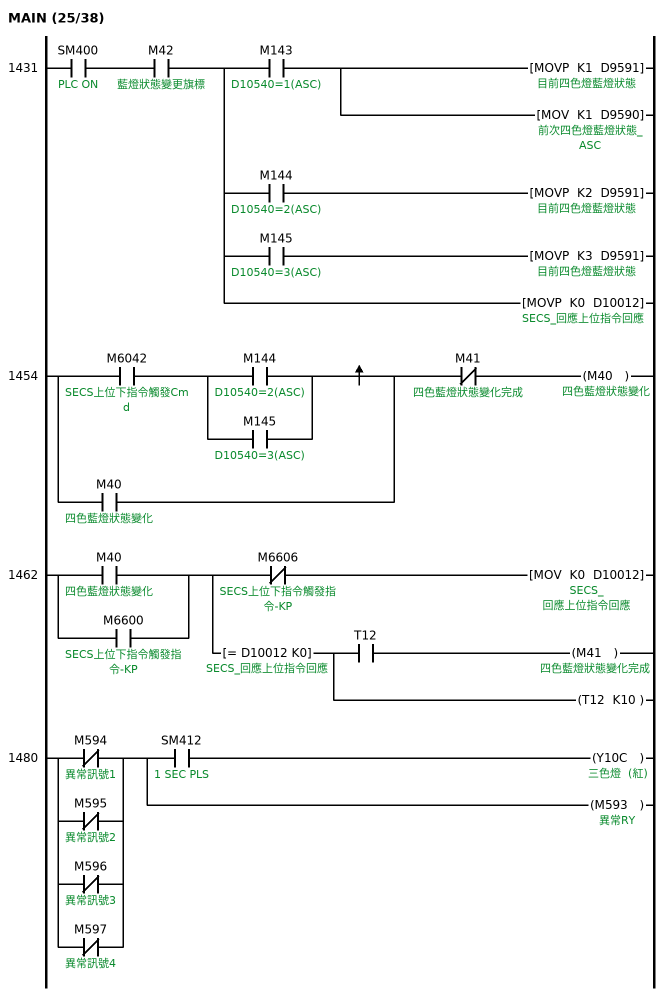
[picture p24: ladder of MAIN, rungs at steps 1431 to 1480]
1431  LD      SM400  ; PLC ON
      AND     M42  ; 藍燈狀態變更旗標
      MPS
      AND     M143  ; D10540=1(ASC)
      MOVP    K1 D9591
      MOV     K1 D9590
      MRD
      AND     M144  ; D10540=2(ASC)
      MOVP    K2 D9591
      MRD
      AND     M145  ; D10540=3(ASC)
      MOVP    K3 D9591
      MPP
      MOVP    K0 D10012  ; SECS_回應上位指令回應
1454  LD      M6042  ; SECS上位下指令觸發Cmd
      LD      M144  ; D10540=2(ASC)
      OR      M145  ; D10540=3(ASC)
      ANB
      MEP
      OR      M40  ; 四色藍燈狀態變化
      ANI     M41  ; 四色藍燈狀態變化完成
      OUT     M40  ; 四色藍燈狀態變化
1462  LD      M40  ; 四色藍燈狀態變化
      OR      M6600  ; SECS上位下指令觸發指令-KP
      MPS
      ANI     M6606  ; SECS上位下指令觸發指令-KP
      MOV     K0 D10012
      MPP
      AND=    D10012 K0  ; SECS_回應上位指令回應
      MPS
      AND     T12
      OUT     M41  ; 四色藍燈狀態變化完成
      MPP
      OUT     T12 K10
1480  LDI     M594  ; 異常訊號1
      ORI     M595  ; 異常訊號2
      ORI     M596  ; 異常訊號3
      ORI     M597  ; 異常訊號4
      MPS
      AND     SM412  ; 1 SEC PLS
      OUT     Y10C  ; 三色燈  (紅)
      MPP
      OUT     M593  ; 異常RY
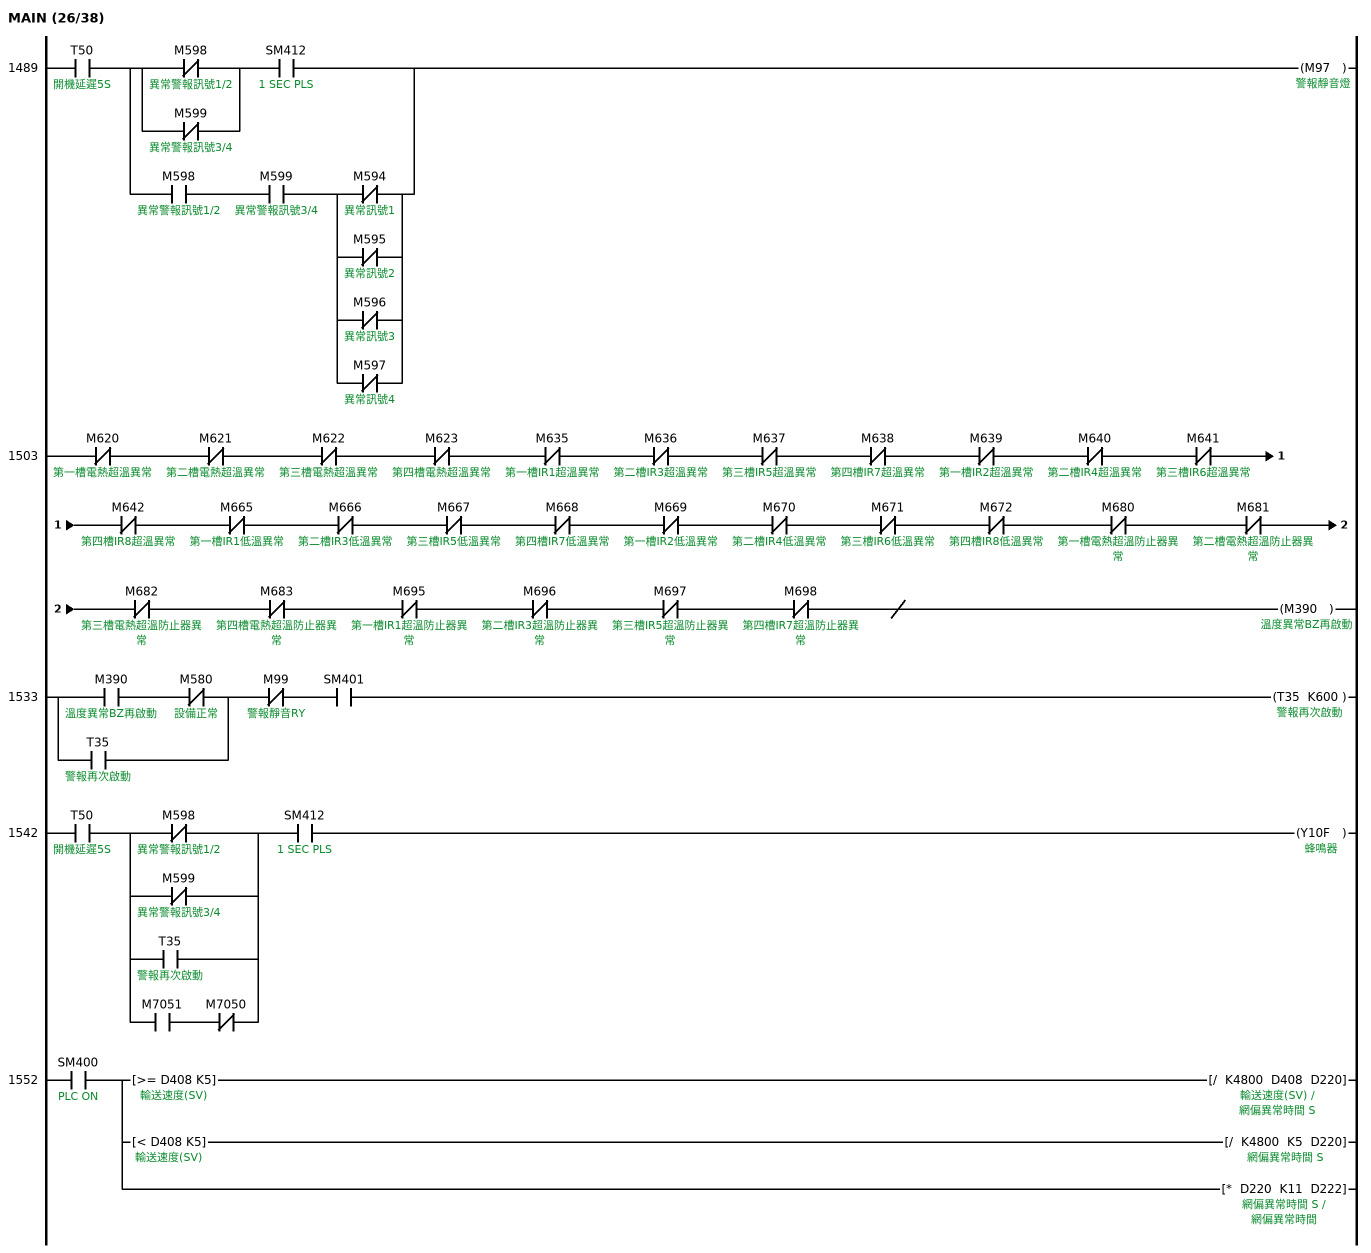
1489  LD      T50  ; 開機延遲5S
      LDI     M598  ; 異常警報訊號1/2
      ORI     M599  ; 異常警報訊號3/4
      AND     SM412  ; 1 SEC PLS
      LD      M598  ; 異常警報訊號1/2
      AND     M599  ; 異常警報訊號3/4
      LDI     M594  ; 異常訊號1
      ORI     M595  ; 異常訊號2
      ORI     M596  ; 異常訊號3
      ORI     M597  ; 異常訊號4
      ANB
      ORB
      ANB
      OUT     M97  ; 警報靜音燈
1503  LDI     M620  ; 第一槽電熱超溫異常
      ANI     M621  ; 第二槽電熱超溫異常
      ANI     M622  ; 第三槽電熱超溫異常
      ANI     M623  ; 第四槽電熱超溫異常
      ANI     M635  ; 第一槽IR1超溫異常
      ANI     M636  ; 第二槽IR3超溫異常
      ANI     M637  ; 第三槽IR5超溫異常
      ANI     M638  ; 第四槽IR7超溫異常
      ANI     M639  ; 第一槽IR2超溫異常
      ANI     M640  ; 第二槽IR4超溫異常
      ANI     M641  ; 第三槽IR6超溫異常
      ANI     M642  ; 第四槽IR8超溫異常
      ANI     M665  ; 第一槽IR1低溫異常
      ANI     M666  ; 第二槽IR3低溫異常
      ANI     M667  ; 第三槽IR5低溫異常
      ANI     M668  ; 第四槽IR7低溫異常
      ANI     M669  ; 第一槽IR2低溫異常
      ANI     M670  ; 第二槽IR4低溫異常
      ANI     M671  ; 第三槽IR6低溫異常
      ANI     M672  ; 第四槽IR8低溫異常
      ANI     M680  ; 第一槽電熱超溫防止器異常
      ANI     M681  ; 第二槽電熱超溫防止器異常
      ANI     M682  ; 第三槽電熱超溫防止器異常
      ANI     M683  ; 第四槽電熱超溫防止器異常
      ANI     M695  ; 第一槽IR1超溫防止器異常
      ANI     M696  ; 第二槽IR3超溫防止器異常
      ANI     M697  ; 第三槽IR5超溫防止器異常
      ANI     M698  ; 第四槽IR7超溫防止器異常
      INV
      OUT     M390  ; 溫度異常BZ再啟動
1533  LD      M390  ; 溫度異常BZ再啟動
      ANI     M580  ; 設備正常
      OR      T35  ; 警報再次啟動
      ANI     M99  ; 警報靜音RY
      AND     SM401
      OUT     T35 K600  ; 警報再次啟動
1542  LD      T50  ; 開機延遲5S
      LDI     M598  ; 異常警報訊號1/2
      ORI     M599  ; 異常警報訊號3/4
      OR      T35  ; 警報再次啟動
      LD      M7051
      ANI     M7050
      ORB
      ANB
      AND     SM412  ; 1 SEC PLS
      OUT     Y10F  ; 蜂鳴器
1552  LD      SM400  ; PLC ON
      MPS
      AND>=   D408 K5  ; 輸送速度(SV)
      /       K4800 D408 D220  ; 網偏異常時間 S
      MRD
      AND<    D408 K5  ; 輸送速度(SV)
      /       K4800 K5 D220
      MPP
      *       D220 K11 D222  ; 網偏異常時間
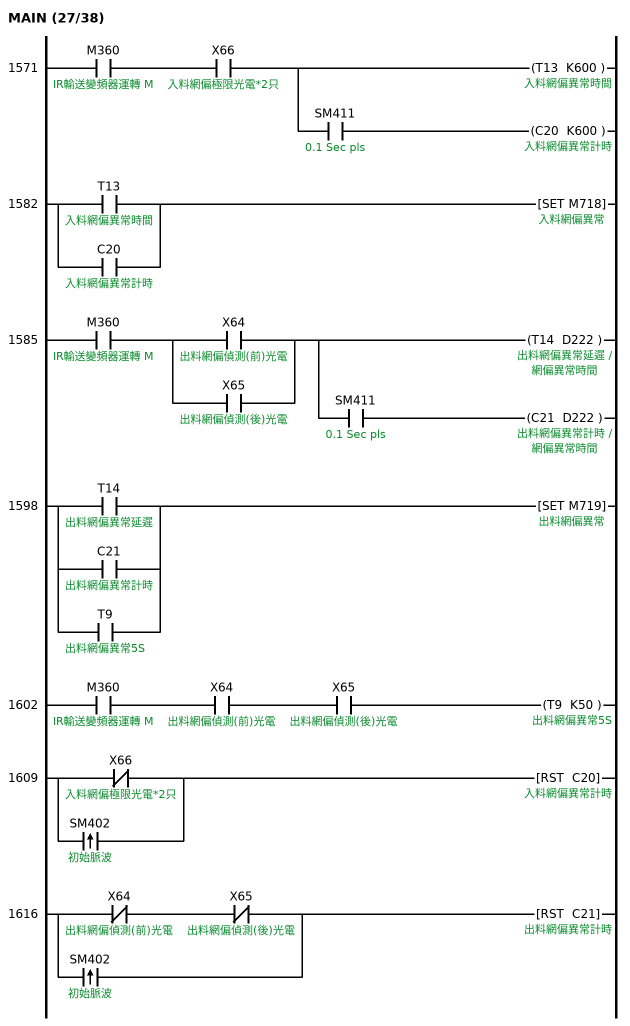
1571  LD      M360  ; IR輸送變頻器運轉 M
      AND     X66  ; 入料網偏極限光電*2只
      OUT     T13 K600  ; 入料網偏異常時間
      AND     SM411  ; 0.1 Sec pls
      OUT     C20 K600  ; 入料網偏異常計時
1582  LD      T13  ; 入料網偏異常時間
      OR      C20  ; 入料網偏異常計時
      SET     M718  ; 入料網偏異常
1585  LD      M360  ; IR輸送變頻器運轉 M
      LD      X64  ; 出料網偏偵測(前)光電
      OR      X65  ; 出料網偏偵測(後)光電
      ANB
      OUT     T14 D222  ; 出料網偏異常延遲 / 網偏異常時間
      AND     SM411  ; 0.1 Sec pls
      OUT     C21 D222  ; 出料網偏異常計時 / 網偏異常時間
1598  LD      T14  ; 出料網偏異常延遲
      OR      C21  ; 出料網偏異常計時
      OR      T9  ; 出料網偏異常5S
      SET     M719  ; 出料網偏異常
1602  LD      M360  ; IR輸送變頻器運轉 M
      AND     X64  ; 出料網偏偵測(前)光電
      AND     X65  ; 出料網偏偵測(後)光電
      OUT     T9 K50  ; 出料網偏異常5S
1609  LDI     X66  ; 入料網偏極限光電*2只
      ORP     SM402  ; 初始脈波
      RST     C20  ; 入料網偏異常計時
1616  LDI     X64  ; 出料網偏偵測(前)光電
      ANI     X65  ; 出料網偏偵測(後)光電
      ORP     SM402  ; 初始脈波
      RST     C21  ; 出料網偏異常計時
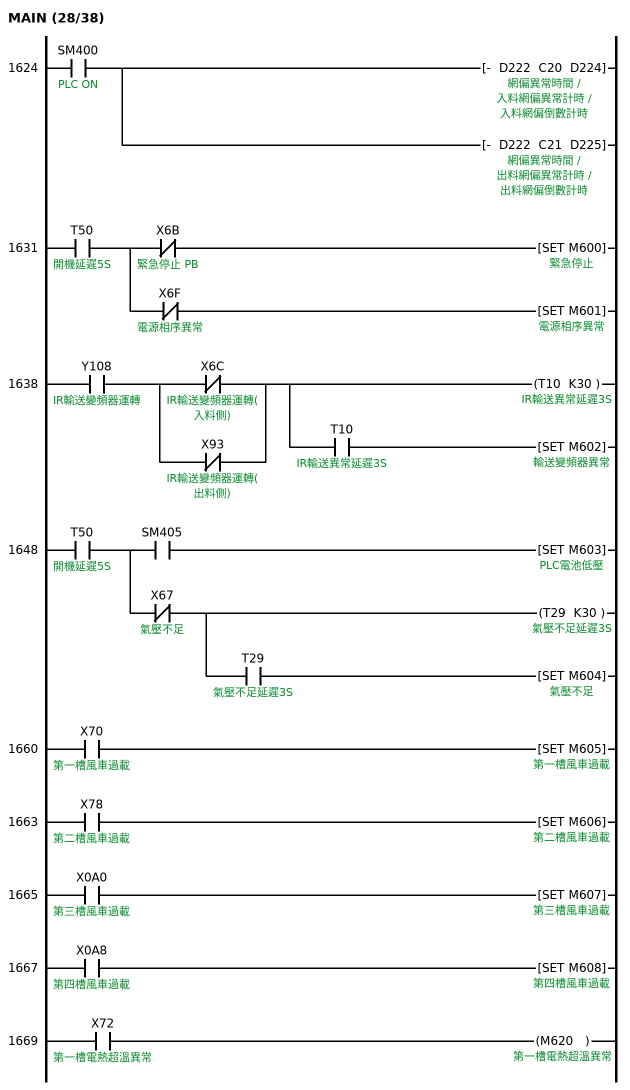
1624  LD      SM400  ; PLC ON
      -       D222 C20 D224  ; 入料網偏倒數計時
      -       D222 C21 D225  ; 出料網偏倒數計時
1631  LD      T50  ; 開機延遲5S
      MPS
      ANI     X6B  ; 緊急停止 PB
      SET     M600  ; 緊急停止
      MPP
      ANI     X6F  ; 電源相序異常
      SET     M601  ; 電源相序異常
1638  LD      Y108  ; IR輸送變頻器運轉
      LDI     X6C  ; IR輸送變頻器運轉(入料側)
      ORI     X93  ; IR輸送變頻器運轉(出料側)
      ANB
      OUT     T10 K30  ; IR輸送異常延遲3S
      AND     T10  ; IR輸送異常延遲3S
      SET     M602  ; 輸送變頻器異常
1648  LD      T50  ; 開機延遲5S
      MPS
      AND     SM405
      SET     M603  ; PLC電池低壓
      MPP
      ANI     X67  ; 氣壓不足
      OUT     T29 K30  ; 氣壓不足延遲3S
      AND     T29  ; 氣壓不足延遲3S
      SET     M604  ; 氣壓不足
1660  LD      X70  ; 第一槽風車過載
      SET     M605  ; 第一槽風車過載
        [note] 
1663  LD      X78  ; 第二槽風車過載
      SET     M606  ; 第二槽風車過載
1665  LD      X0A0  ; 第三槽風車過載
      SET     M607  ; 第三槽風車過載
1667  LD      X0A8  ; 第四槽風車過載
      SET     M608  ; 第四槽風車過載
1669  LD      X72  ; 第一槽電熱超溫異常
      OUT     M620  ; 第一槽電熱超溫異常
        [note] 
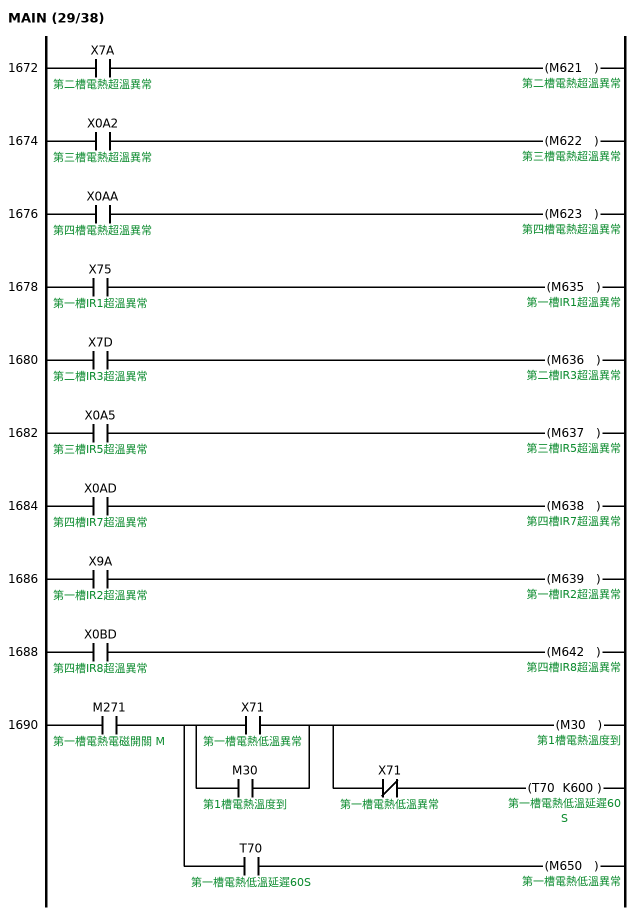
1672  LD      X7A  ; 第二槽電熱超溫異常
      OUT     M621  ; 第二槽電熱超溫異常
1674  LD      X0A2  ; 第三槽電熱超溫異常
      OUT     M622  ; 第三槽電熱超溫異常
1676  LD      X0AA  ; 第四槽電熱超溫異常
      OUT     M623  ; 第四槽電熱超溫異常
1678  LD      X75  ; 第一槽IR1超溫異常
      OUT     M635  ; 第一槽IR1超溫異常
1680  LD      X7D  ; 第二槽IR3超溫異常
      OUT     M636  ; 第二槽IR3超溫異常
1682  LD      X0A5  ; 第三槽IR5超溫異常
      OUT     M637  ; 第三槽IR5超溫異常
1684  LD      X0AD  ; 第四槽IR7超溫異常
      OUT     M638  ; 第四槽IR7超溫異常
1686  LD      X9A  ; 第一槽IR2超溫異常
      OUT     M639  ; 第一槽IR2超溫異常
1688  LD      X0BD  ; 第四槽IR8超溫異常
      OUT     M642  ; 第四槽IR8超溫異常
1690  LD      M271  ; 第一槽電熱電磁開關 M
      MPS
      LD      X71  ; 第一槽電熱低溫異常
      OR      M30  ; 第1槽電熱溫度到
      ANB
      OUT     M30  ; 第1槽電熱溫度到
        [note] 
      ANI     X71  ; 第一槽電熱低溫異常
      OUT     T70 K600  ; 第一槽電熱低溫延遲60S
      MPP
      AND     T70  ; 第一槽電熱低溫延遲60S
      OUT     M650  ; 第一槽電熱低溫異常
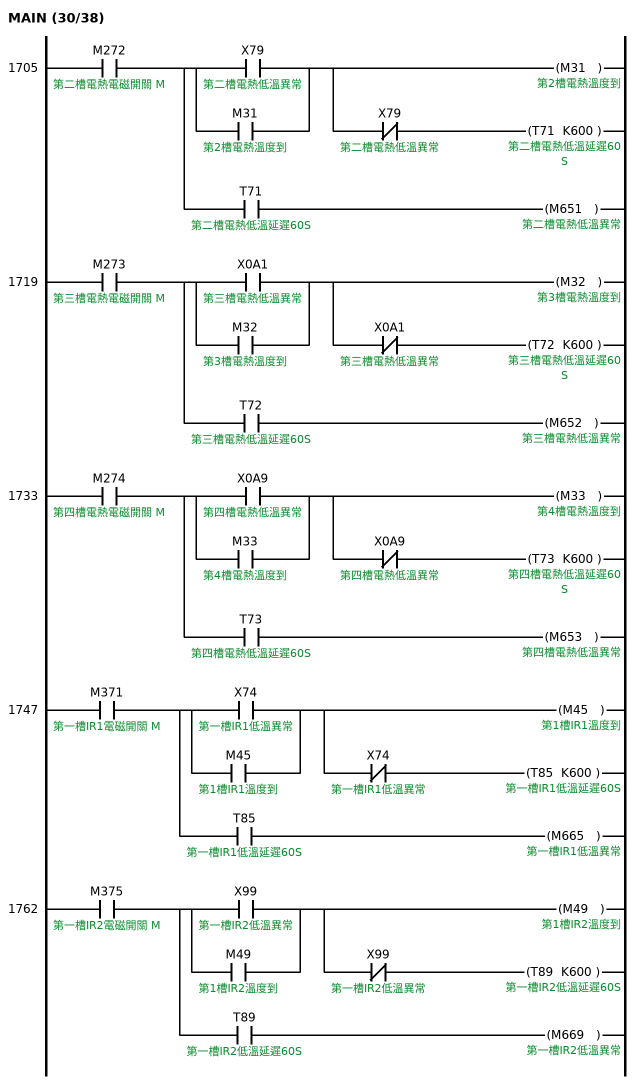
1705  LD      M272  ; 第二槽電熱電磁開關 M
      MPS
      LD      X79  ; 第二槽電熱低溫異常
      OR      M31  ; 第2槽電熱溫度到
      ANB
      OUT     M31  ; 第2槽電熱溫度到
      ANI     X79  ; 第二槽電熱低溫異常
      OUT     T71 K600  ; 第二槽電熱低溫延遲60S
      MPP
      AND     T71  ; 第二槽電熱低溫延遲60S
      OUT     M651  ; 第二槽電熱低溫異常
1719  LD      M273  ; 第三槽電熱電磁開關 M
      MPS
      LD      X0A1  ; 第三槽電熱低溫異常
      OR      M32  ; 第3槽電熱溫度到
      ANB
      OUT     M32  ; 第3槽電熱溫度到
      ANI     X0A1  ; 第三槽電熱低溫異常
      OUT     T72 K600  ; 第三槽電熱低溫延遲60S
      MPP
      AND     T72  ; 第三槽電熱低溫延遲60S
      OUT     M652  ; 第三槽電熱低溫異常
1733  LD      M274  ; 第四槽電熱電磁開關 M
      MPS
      LD      X0A9  ; 第四槽電熱低溫異常
      OR      M33  ; 第4槽電熱溫度到
      ANB
      OUT     M33  ; 第4槽電熱溫度到
      ANI     X0A9  ; 第四槽電熱低溫異常
      OUT     T73 K600  ; 第四槽電熱低溫延遲60S
      MPP
      AND     T73  ; 第四槽電熱低溫延遲60S
      OUT     M653  ; 第四槽電熱低溫異常
1747  LD      M371  ; 第一槽IR1電磁開關 M
      MPS
      LD      X74  ; 第一槽IR1低溫異常
      OR      M45  ; 第1槽IR1溫度到
      ANB
      OUT     M45  ; 第1槽IR1溫度到
        [note] 
      ANI     X74  ; 第一槽IR1低溫異常
      OUT     T85 K600  ; 第一槽IR1低溫延遲60S
      MPP
      AND     T85  ; 第一槽IR1低溫延遲60S
      OUT     M665  ; 第一槽IR1低溫異常
1762  LD      M375  ; 第一槽IR2電磁開關 M
      MPS
      LD      X99  ; 第一槽IR2低溫異常
      OR      M49  ; 第1槽IR2溫度到
      ANB
      OUT     M49  ; 第1槽IR2溫度到
      ANI     X99  ; 第一槽IR2低溫異常
      OUT     T89 K600  ; 第一槽IR2低溫延遲60S
      MPP
      AND     T89  ; 第一槽IR2低溫延遲60S
      OUT     M669  ; 第一槽IR2低溫異常
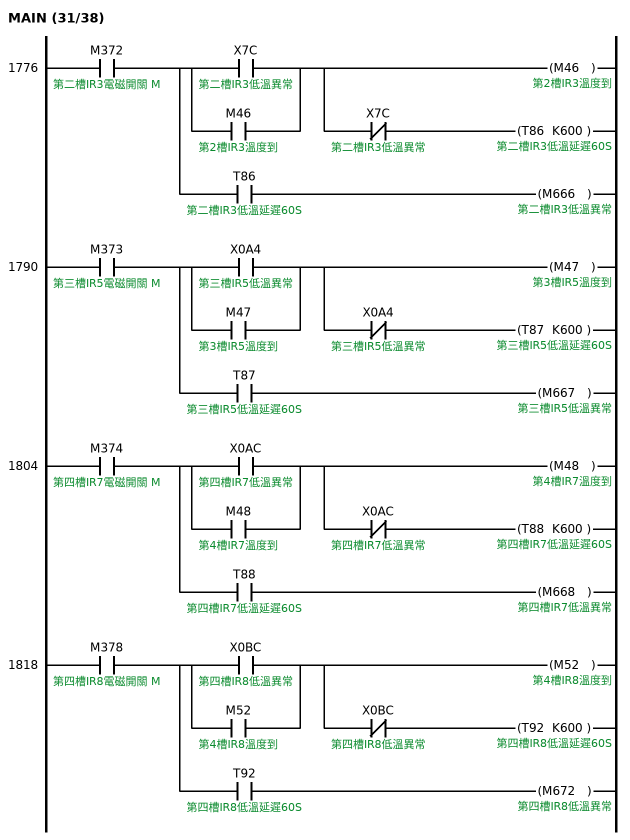
1776  LD      M372  ; 第二槽IR3電磁開關 M
      MPS
      LD      X7C  ; 第二槽IR3低溫異常
      OR      M46  ; 第2槽IR3溫度到
      ANB
      OUT     M46  ; 第2槽IR3溫度到
      ANI     X7C  ; 第二槽IR3低溫異常
      OUT     T86 K600  ; 第二槽IR3低溫延遲60S
      MPP
      AND     T86  ; 第二槽IR3低溫延遲60S
      OUT     M666  ; 第二槽IR3低溫異常
1790  LD      M373  ; 第三槽IR5電磁開關 M
      MPS
      LD      X0A4  ; 第三槽IR5低溫異常
      OR      M47  ; 第3槽IR5溫度到
      ANB
      OUT     M47  ; 第3槽IR5溫度到
      ANI     X0A4  ; 第三槽IR5低溫異常
      OUT     T87 K600  ; 第三槽IR5低溫延遲60S
      MPP
      AND     T87  ; 第三槽IR5低溫延遲60S
      OUT     M667  ; 第三槽IR5低溫異常
1804  LD      M374  ; 第四槽IR7電磁開關 M
      MPS
      LD      X0AC  ; 第四槽IR7低溫異常
      OR      M48  ; 第4槽IR7溫度到
      ANB
      OUT     M48  ; 第4槽IR7溫度到
      ANI     X0AC  ; 第四槽IR7低溫異常
      OUT     T88 K600  ; 第四槽IR7低溫延遲60S
      MPP
      AND     T88  ; 第四槽IR7低溫延遲60S
      OUT     M668  ; 第四槽IR7低溫異常
1818  LD      M378  ; 第四槽IR8電磁開關 M
      MPS
      LD      X0BC  ; 第四槽IR8低溫異常
      OR      M52  ; 第4槽IR8溫度到
      ANB
      OUT     M52  ; 第4槽IR8溫度到
      ANI     X0BC  ; 第四槽IR8低溫異常
      OUT     T92 K600  ; 第四槽IR8低溫延遲60S
      MPP
      AND     T92  ; 第四槽IR8低溫延遲60S
      OUT     M672  ; 第四槽IR8低溫異常
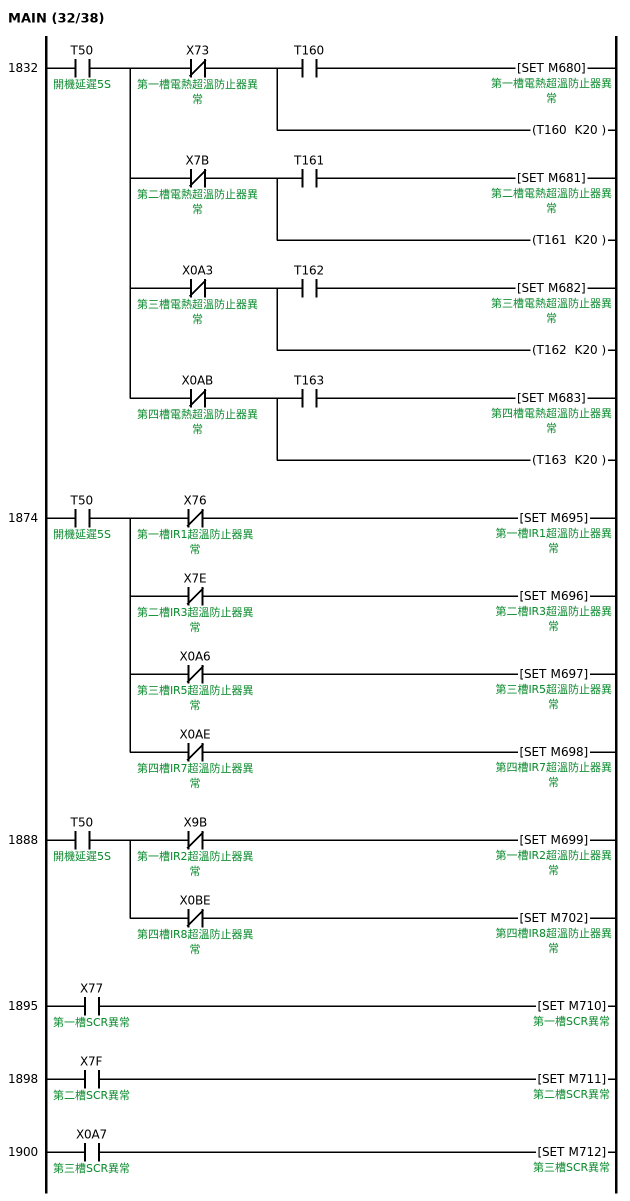
1832  LD      T50  ; 開機延遲5S
      MPS
      ANI     X73  ; 第一槽電熱超溫防止器異常
      MPS
      AND     T160
      SET     M680  ; 第一槽電熱超溫防止器異常
        [note] 
      MPP
      OUT     T160 K20
      MRD
      ANI     X7B  ; 第二槽電熱超溫防止器異常
      MPS
      AND     T161
      SET     M681  ; 第二槽電熱超溫防止器異常
      MPP
      OUT     T161 K20
      MRD
      ANI     X0A3  ; 第三槽電熱超溫防止器異常
      MPS
      AND     T162
      SET     M682  ; 第三槽電熱超溫防止器異常
      MPP
      OUT     T162 K20
      MPP
      ANI     X0AB  ; 第四槽電熱超溫防止器異常
      MPS
      AND     T163
      SET     M683  ; 第四槽電熱超溫防止器異常
      MPP
      OUT     T163 K20
1874  LD      T50  ; 開機延遲5S
      MPS
      ANI     X76  ; 第一槽IR1超溫防止器異常
      SET     M695  ; 第一槽IR1超溫防止器異常
        [note] 
      MRD
      ANI     X7E  ; 第二槽IR3超溫防止器異常
      SET     M696  ; 第二槽IR3超溫防止器異常
      MRD
      ANI     X0A6  ; 第三槽IR5超溫防止器異常
      SET     M697  ; 第三槽IR5超溫防止器異常
      MPP
      ANI     X0AE  ; 第四槽IR7超溫防止器異常
      SET     M698  ; 第四槽IR7超溫防止器異常
1888  LD      T50  ; 開機延遲5S
      MPS
      ANI     X9B  ; 第一槽IR2超溫防止器異常
      SET     M699  ; 第一槽IR2超溫防止器異常
      MPP
      ANI     X0BE  ; 第四槽IR8超溫防止器異常
      SET     M702  ; 第四槽IR8超溫防止器異常
1895  LD      X77  ; 第一槽SCR異常
      SET     M710  ; 第一槽SCR異常
        [note] 
1898  LD      X7F  ; 第二槽SCR異常
      SET     M711  ; 第二槽SCR異常
1900  LD      X0A7  ; 第三槽SCR異常
      SET     M712  ; 第三槽SCR異常
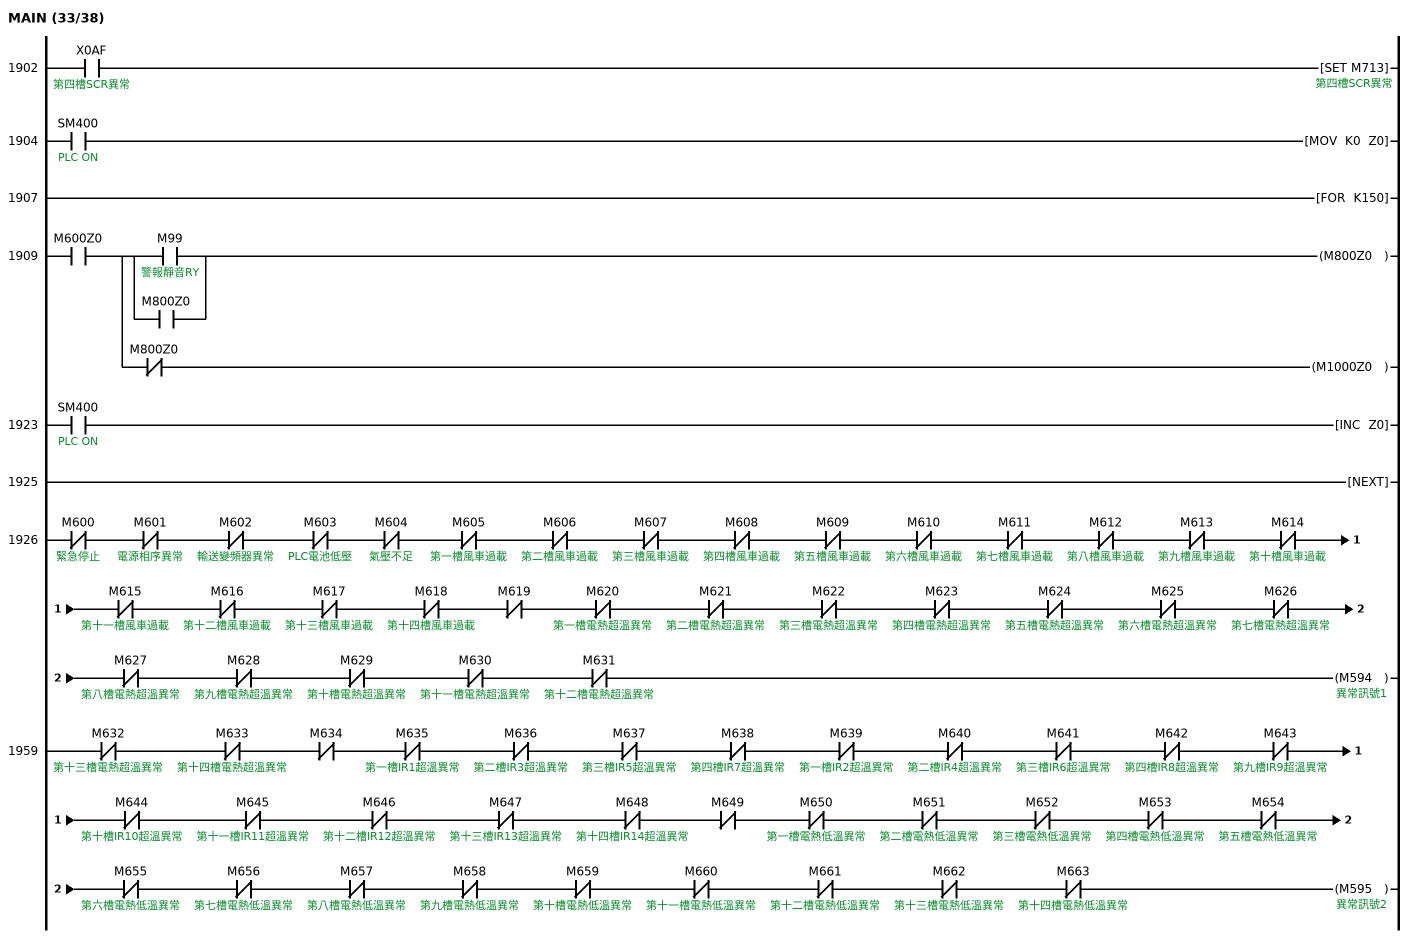
1902  LD      X0AF  ; 第四槽SCR異常
      SET     M713  ; 第四槽SCR異常
1904  LD      SM400  ; PLC ON
      MOV     K0 Z0
1907  FOR     K150
1909  LD      M600Z0
      MPS
      LD      M99  ; 警報靜音RY
      OR      M800Z0
      ANB
      OUT     M800Z0
      MPP
      ANI     M800Z0
      OUT     M1000Z0
1923  LD      SM400  ; PLC ON
      INC     Z0
1925  NEXT
1926  LDI     M600  ; 緊急停止
      ANI     M601  ; 電源相序異常
      ANI     M602  ; 輸送變頻器異常
      ANI     M603  ; PLC電池低壓
      ANI     M604  ; 氣壓不足
      ANI     M605  ; 第一槽風車過載
      ANI     M606  ; 第二槽風車過載
      ANI     M607  ; 第三槽風車過載
      ANI     M608  ; 第四槽風車過載
      ANI     M609  ; 第五槽風車過載
      ANI     M610  ; 第六槽風車過載
      ANI     M611  ; 第七槽風車過載
      ANI     M612  ; 第八槽風車過載
      ANI     M613  ; 第九槽風車過載
      ANI     M614  ; 第十槽風車過載
      ANI     M615  ; 第十一槽風車過載
      ANI     M616  ; 第十二槽風車過載
      ANI     M617  ; 第十三槽風車過載
      ANI     M618  ; 第十四槽風車過載
      ANI     M619
      ANI     M620  ; 第一槽電熱超溫異常
      ANI     M621  ; 第二槽電熱超溫異常
      ANI     M622  ; 第三槽電熱超溫異常
      ANI     M623  ; 第四槽電熱超溫異常
      ANI     M624  ; 第五槽電熱超溫異常
      ANI     M625  ; 第六槽電熱超溫異常
      ANI     M626  ; 第七槽電熱超溫異常
      ANI     M627  ; 第八槽電熱超溫異常
      ANI     M628  ; 第九槽電熱超溫異常
      ANI     M629  ; 第十槽電熱超溫異常
      ANI     M630  ; 第十一槽電熱超溫異常
      ANI     M631  ; 第十二槽電熱超溫異常
      OUT     M594  ; 異常訊號1
1959  LDI     M632  ; 第十三槽電熱超溫異常
      ANI     M633  ; 第十四槽電熱超溫異常
      ANI     M634
      ANI     M635  ; 第一槽IR1超溫異常
      ANI     M636  ; 第二槽IR3超溫異常
      ANI     M637  ; 第三槽IR5超溫異常
      ANI     M638  ; 第四槽IR7超溫異常
      ANI     M639  ; 第一槽IR2超溫異常
      ANI     M640  ; 第二槽IR4超溫異常
      ANI     M641  ; 第三槽IR6超溫異常
      ANI     M642  ; 第四槽IR8超溫異常
      ANI     M643  ; 第九槽IR9超溫異常
      ANI     M644  ; 第十槽IR10超溫異常
      ANI     M645  ; 第十一槽IR11超溫異常
      ANI     M646  ; 第十二槽IR12超溫異常
      ANI     M647  ; 第十三槽IR13超溫異常
      ANI     M648  ; 第十四槽IR14超溫異常
      ANI     M649
      ANI     M650  ; 第一槽電熱低溫異常
      ANI     M651  ; 第二槽電熱低溫異常
      ANI     M652  ; 第三槽電熱低溫異常
      ANI     M653  ; 第四槽電熱低溫異常
      ANI     M654  ; 第五槽電熱低溫異常
      ANI     M655  ; 第六槽電熱低溫異常
      ANI     M656  ; 第七槽電熱低溫異常
      ANI     M657  ; 第八槽電熱低溫異常
      ANI     M658  ; 第九槽電熱低溫異常
      ANI     M659  ; 第十槽電熱低溫異常
      ANI     M660  ; 第十一槽電熱低溫異常
      ANI     M661  ; 第十二槽電熱低溫異常
      ANI     M662  ; 第十三槽電熱低溫異常
      ANI     M663  ; 第十四槽電熱低溫異常
      OUT     M595  ; 異常訊號2
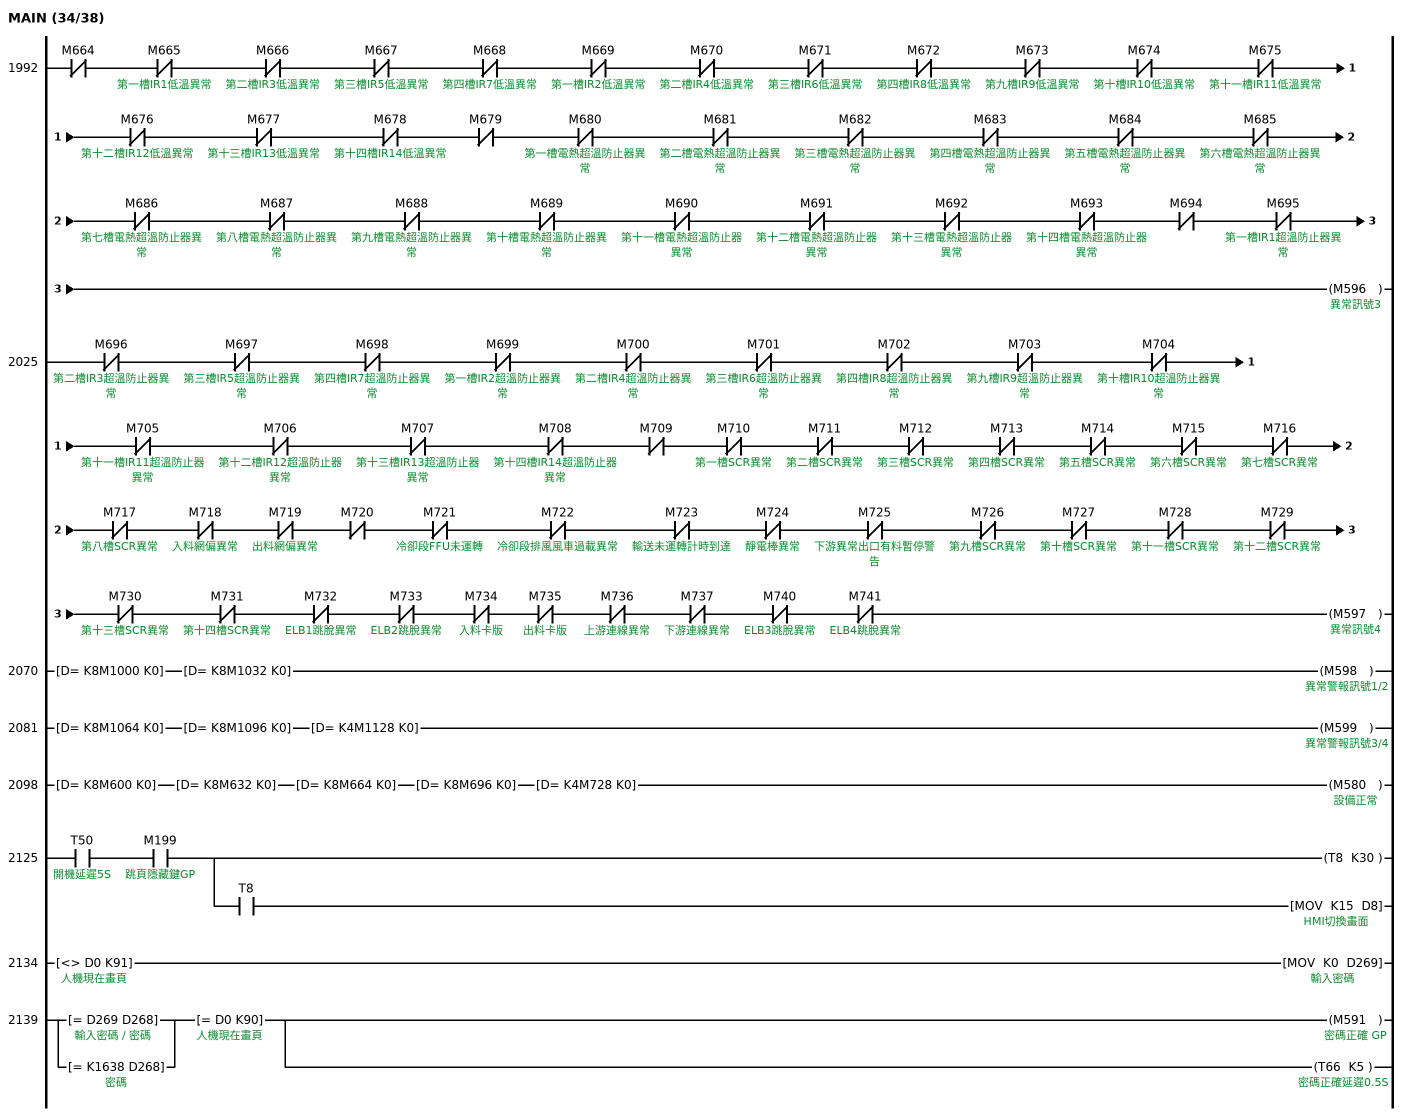
1992  LDI     M664
      ANI     M665  ; 第一槽IR1低溫異常
      ANI     M666  ; 第二槽IR3低溫異常
      ANI     M667  ; 第三槽IR5低溫異常
      ANI     M668  ; 第四槽IR7低溫異常
      ANI     M669  ; 第一槽IR2低溫異常
      ANI     M670  ; 第二槽IR4低溫異常
      ANI     M671  ; 第三槽IR6低溫異常
      ANI     M672  ; 第四槽IR8低溫異常
      ANI     M673  ; 第九槽IR9低溫異常
      ANI     M674  ; 第十槽IR10低溫異常
      ANI     M675  ; 第十一槽IR11低溫異常
      ANI     M676  ; 第十二槽IR12低溫異常
      ANI     M677  ; 第十三槽IR13低溫異常
      ANI     M678  ; 第十四槽IR14低溫異常
      ANI     M679
      ANI     M680  ; 第一槽電熱超溫防止器異常
      ANI     M681  ; 第二槽電熱超溫防止器異常
      ANI     M682  ; 第三槽電熱超溫防止器異常
      ANI     M683  ; 第四槽電熱超溫防止器異常
      ANI     M684  ; 第五槽電熱超溫防止器異常
      ANI     M685  ; 第六槽電熱超溫防止器異常
      ANI     M686  ; 第七槽電熱超溫防止器異常
      ANI     M687  ; 第八槽電熱超溫防止器異常
      ANI     M688  ; 第九槽電熱超溫防止器異常
      ANI     M689  ; 第十槽電熱超溫防止器異常
      ANI     M690  ; 第十一槽電熱超溫防止器異常
      ANI     M691  ; 第十二槽電熱超溫防止器異常
      ANI     M692  ; 第十三槽電熱超溫防止器異常
      ANI     M693  ; 第十四槽電熱超溫防止器異常
      ANI     M694
      ANI     M695  ; 第一槽IR1超溫防止器異常
      OUT     M596  ; 異常訊號3
2025  LDI     M696  ; 第二槽IR3超溫防止器異常
      ANI     M697  ; 第三槽IR5超溫防止器異常
      ANI     M698  ; 第四槽IR7超溫防止器異常
      ANI     M699  ; 第一槽IR2超溫防止器異常
      ANI     M700  ; 第二槽IR4超溫防止器異常
      ANI     M701  ; 第三槽IR6超溫防止器異常
      ANI     M702  ; 第四槽IR8超溫防止器異常
      ANI     M703  ; 第九槽IR9超溫防止器異常
      ANI     M704  ; 第十槽IR10超溫防止器異常
      ANI     M705  ; 第十一槽IR11超溫防止器異常
      ANI     M706  ; 第十二槽IR12超溫防止器異常
      ANI     M707  ; 第十三槽IR13超溫防止器異常
      ANI     M708  ; 第十四槽IR14超溫防止器異常
      ANI     M709
      ANI     M710  ; 第一槽SCR異常
      ANI     M711  ; 第二槽SCR異常
      ANI     M712  ; 第三槽SCR異常
      ANI     M713  ; 第四槽SCR異常
      ANI     M714  ; 第五槽SCR異常
      ANI     M715  ; 第六槽SCR異常
      ANI     M716  ; 第七槽SCR異常
      ANI     M717  ; 第八槽SCR異常
      ANI     M718  ; 入料網偏異常
      ANI     M719  ; 出料網偏異常
      ANI     M720
      ANI     M721  ; 冷卻段FFU未運轉
      ANI     M722  ; 冷卻段排風風車過載異常
      ANI     M723  ; 輸送未運轉計時到達
      ANI     M724  ; 靜電棒異常
      ANI     M725  ; 下游異常出口有料暫停警告
      ANI     M726  ; 第九槽SCR異常
      ANI     M727  ; 第十槽SCR異常
      ANI     M728  ; 第十一槽SCR異常
      ANI     M729  ; 第十二槽SCR異常
      ANI     M730  ; 第十三槽SCR異常
      ANI     M731  ; 第十四槽SCR異常
      ANI     M732  ; ELB1跳脫異常
      ANI     M733  ; ELB2跳脫異常
      ANI     M734  ; 入料卡版
      ANI     M735  ; 出料卡版
      ANI     M736  ; 上游連線異常
      ANI     M737  ; 下游連線異常
      ANI     M740  ; ELB3跳脫異常
      ANI     M741  ; ELB4跳脫異常
      OUT     M597  ; 異常訊號4
2070  LDD=    K8M1000 K0  ; 緊急停止迴圈資料
      ANDD=   K8M1032 K0  ; 迴圈資料
      OUT     M598  ; 異常警報訊號1/2
2081  LDD=    K8M1064 K0  ; 迴圈資料
      ANDD=   K8M1096 K0  ; 迴圈資料
      ANDD=   K4M1128 K0
      OUT     M599  ; 異常警報訊號3/4
2098  LDD=    K8M600 K0  ; 緊急停止
      ANDD=   K8M632 K0  ; 第十三槽電熱超溫異常
      ANDD=   K8M664 K0
      ANDD=   K8M696 K0  ; 第二槽IR3超溫防止器異常
      ANDD=   K4M728 K0  ; 第十一槽SCR異常
      OUT     M580  ; 設備正常
2125  LD      T50  ; 開機延遲5S
      AND     M199  ; 跳頁隱藏鍵GP
      OUT     T8 K30
      AND     T8
      MOV     K15 D8  ; HMI切換畫面
2134  LD<>    D0 K91  ; 人機現在畫頁
      MOV     K0 D269  ; 輸入密碼
2139  LD=     D269 D268  ; 輸入密碼 / 密碼
      OR=     K1638 D268  ; 密碼
      AND=    D0 K90  ; 人機現在畫頁
      OUT     M591  ; 密碼正確 GP
      OUT     T66 K5  ; 密碼正確延遲0.5S
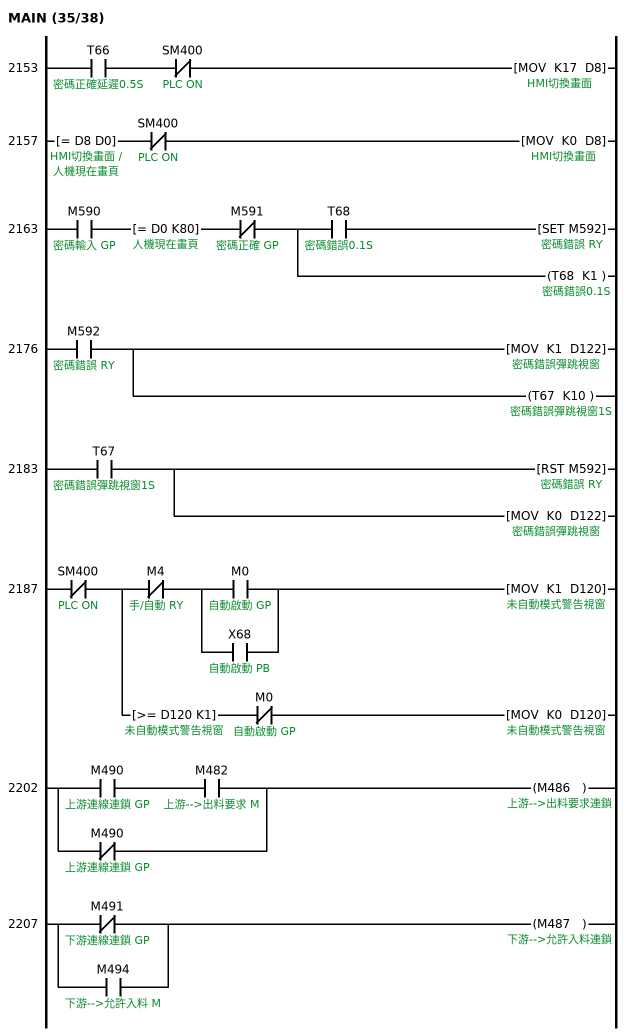
2153  LD      T66  ; 密碼正確延遲0.5S
      ANI     SM400  ; PLC ON
      MOV     K17 D8
2157  LD=     D8 D0  ; HMI切換畫面 / 人機現在畫頁
      ANI     SM400  ; PLC ON
      MOV     K0 D8
2163  LD      M590  ; 密碼輸入 GP
      AND=    D0 K80  ; 人機現在畫頁
      ANI     M591  ; 密碼正確 GP
      MPS
      AND     T68  ; 密碼錯誤0.1S
      SET     M592  ; 密碼錯誤 RY
      MPP
      OUT     T68 K1  ; 密碼錯誤0.1S
2176  LD      M592  ; 密碼錯誤 RY
      MOV     K1 D122  ; 密碼錯誤彈跳視窗
      OUT     T67 K10  ; 密碼錯誤彈跳視窗1S
2183  LD      T67  ; 密碼錯誤彈跳視窗1S
      RST     M592  ; 密碼錯誤 RY
      MOV     K0 D122
2187  LDI     SM400  ; PLC ON
      MPS
      ANI     M4  ; 手/自動 RY
      LD      M0  ; 自動啟動 GP
      OR      X68  ; 自動啟動 PB
      ANB
      MOV     K1 D120  ; 未自動模式警告視窗
      MPP
      AND>=   D120 K1  ; 未自動模式警告視窗
      ANI     M0  ; 自動啟動 GP
      MOV     K0 D120
2202  LD      M490  ; 上游連線連鎖 GP
      AND     M482  ; 上游-->出料要求 M
      ORI     M490  ; 上游連線連鎖 GP
      OUT     M486  ; 上游-->出料要求連鎖
        [note] 
2207  LDI     M491  ; 下游連線連鎖 GP
      OR      M494  ; 下游-->允許入料 M
      OUT     M487  ; 下游-->允許入料連鎖
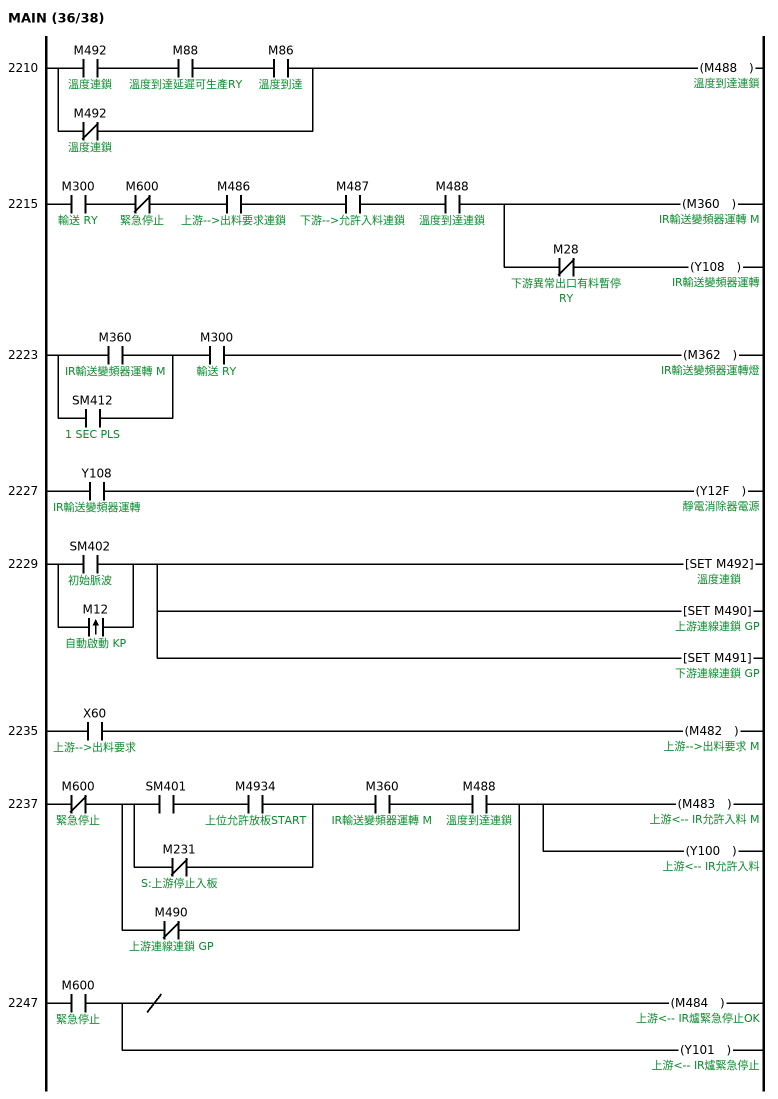
2210  LD      M492  ; 溫度連鎖
      AND     M88  ; 溫度到達延遲可生產RY
      AND     M86  ; 溫度到達
      ORI     M492  ; 溫度連鎖
      OUT     M488  ; 溫度到達連鎖
2215  LD      M300  ; 輸送 RY
      ANI     M600  ; 緊急停止
      AND     M486  ; 上游-->出料要求連鎖
      AND     M487  ; 下游-->允許入料連鎖
      AND     M488  ; 溫度到達連鎖
      OUT     M360  ; IR輸送變頻器運轉 M
      ANI     M28  ; 下游異常出口有料暫停 RY
      OUT     Y108  ; IR輸送變頻器運轉
2223  LD      M360  ; IR輸送變頻器運轉 M
      OR      SM412  ; 1 SEC PLS
      AND     M300  ; 輸送 RY
      OUT     M362  ; IR輸送變頻器運轉燈
2227  LD      Y108  ; IR輸送變頻器運轉
      OUT     Y12F  ; 靜電消除器電源
2229  LD      SM402  ; 初始脈波
      ORP     M12  ; 自動啟動 KP
      SET     M492  ; 溫度連鎖
      SET     M490  ; 上游連線連鎖 GP
      SET     M491  ; 下游連線連鎖 GP
2235  LD      X60  ; 上游-->出料要求
      OUT     M482  ; 上游-->出料要求 M
2237  LDI     M600  ; 緊急停止
      LD      SM401
      AND     M4934  ; 上位允許放板START
      ORI     M231  ; S:上游停止入板
      AND     M360  ; IR輸送變頻器運轉 M
      AND     M488  ; 溫度到達連鎖
      ORI     M490  ; 上游連線連鎖 GP
      ANB
      OUT     M483  ; 上游<-- IR允許入料 M
      OUT     Y100  ; 上游<-- IR允許入料
2247  LD      M600  ; 緊急停止
      MPS
      INV
      OUT     M484  ; 上游<-- IR爐緊急停止OK
      MPP
      OUT     Y101  ; 上游<-- IR爐緊急停止
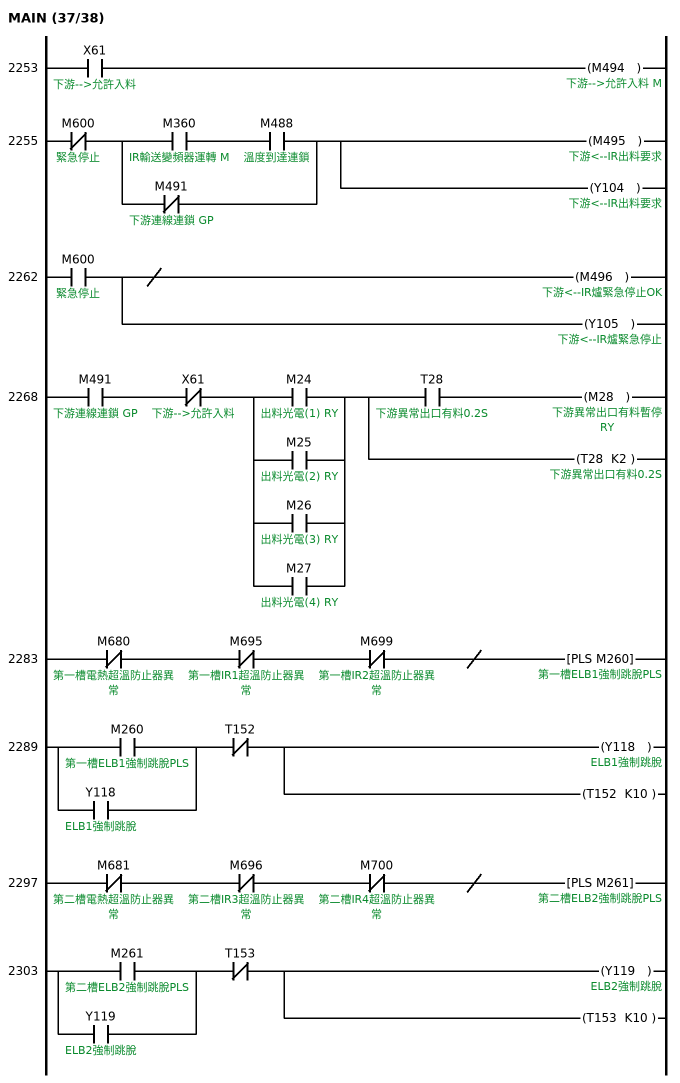
2253  LD      X61  ; 下游-->允許入料
      OUT     M494  ; 下游-->允許入料 M
2255  LDI     M600  ; 緊急停止
      LD      M360  ; IR輸送變頻器運轉 M
      AND     M488  ; 溫度到達連鎖
      ORI     M491  ; 下游連線連鎖 GP
      ANB
      OUT     M495  ; 下游<--IR出料要求
      OUT     Y104  ; 下游<--IR出料要求
2262  LD      M600  ; 緊急停止
      MPS
      INV
      OUT     M496  ; 下游<--IR爐緊急停止OK
      MPP
      OUT     Y105  ; 下游<--IR爐緊急停止
2268  LD      M491  ; 下游連線連鎖 GP
      ANI     X61  ; 下游-->允許入料
      LD      M24  ; 出料光電(1) RY
      OR      M25  ; 出料光電(2) RY
      OR      M26  ; 出料光電(3) RY
      OR      M27  ; 出料光電(4) RY
      ANB
      MPS
      AND     T28  ; 下游異常出口有料0.2S
      OUT     M28  ; 下游異常出口有料暫停 RY
      MPP
      OUT     T28 K2  ; 下游異常出口有料0.2S
2283  LDI     M680  ; 第一槽電熱超溫防止器異常
      ANI     M695  ; 第一槽IR1超溫防止器異常
      ANI     M699  ; 第一槽IR2超溫防止器異常
      INV
      PLS     M260  ; 第一槽ELB1強制跳脫PLS
2289  LD      M260  ; 第一槽ELB1強制跳脫PLS
      OR      Y118  ; ELB1強制跳脫
      ANI     T152
      OUT     Y118  ; ELB1強制跳脫
      OUT     T152 K10
2297  LDI     M681  ; 第二槽電熱超溫防止器異常
      ANI     M696  ; 第二槽IR3超溫防止器異常
      ANI     M700  ; 第二槽IR4超溫防止器異常
      INV
      PLS     M261  ; 第二槽ELB2強制跳脫PLS
2303  LD      M261  ; 第二槽ELB2強制跳脫PLS
      OR      Y119  ; ELB2強制跳脫
      ANI     T153
      OUT     Y119  ; ELB2強制跳脫
      OUT     T153 K10
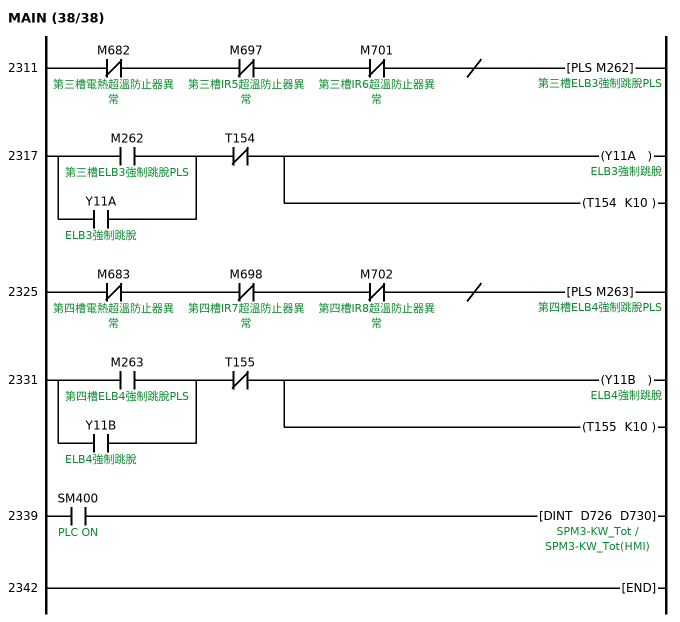
2311  LDI     M682  ; 第三槽電熱超溫防止器異常
      ANI     M697  ; 第三槽IR5超溫防止器異常
      ANI     M701  ; 第三槽IR6超溫防止器異常
      INV
      PLS     M262  ; 第三槽ELB3強制跳脫PLS
2317  LD      M262  ; 第三槽ELB3強制跳脫PLS
      OR      Y11A  ; ELB3強制跳脫
      ANI     T154
      OUT     Y11A  ; ELB3強制跳脫
      OUT     T154 K10
2325  LDI     M683  ; 第四槽電熱超溫防止器異常
      ANI     M698  ; 第四槽IR7超溫防止器異常
      ANI     M702  ; 第四槽IR8超溫防止器異常
      INV
      PLS     M263  ; 第四槽ELB4強制跳脫PLS
2331  LD      M263  ; 第四槽ELB4強制跳脫PLS
      OR      Y11B  ; ELB4強制跳脫
      ANI     T155
      OUT     Y11B  ; ELB4強制跳脫
      OUT     T155 K10
2339  LD      SM400  ; PLC ON
      DINT    D726 D730  ; SPM3-KW_Tot / SPM3-KW_Tot(HMI)
2342  END
END_PROGRAM

PROGRAM SECS
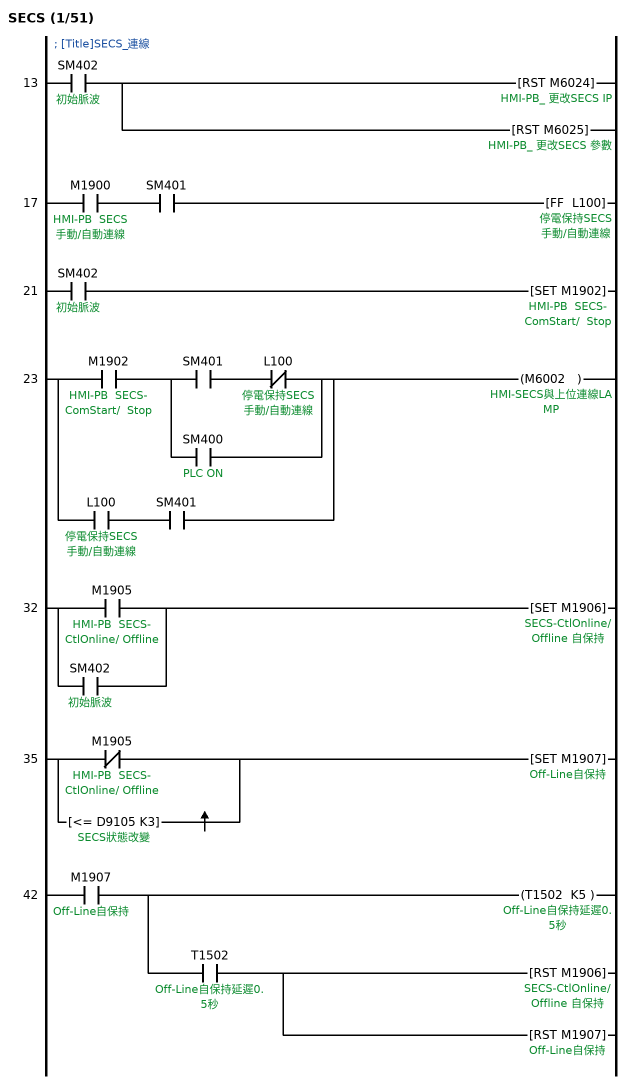
; [Title]SECS_連線
13    LD      SM402  ; 初始脈波
      RST     M6024  ; HMI-PB_ 更改SECS IP
      RST     M6025  ; HMI-PB_ 更改SECS 參數
17    LD      M1900  ; HMI-PB  SECS    手動/自動連線
      AND     SM401
      FF      L100  ; 停電保持SECS    手動/自動連線
21    LD      SM402  ; 初始脈波
      SET     M1902  ; HMI-PB  SECS-ComStart/  Stop
23    LD      M1902  ; HMI-PB  SECS-ComStart/  Stop
      LD      SM401
      ANI     L100  ; 停電保持SECS    手動/自動連線
      OR      SM400  ; PLC ON
      ANB
      LD      L100  ; 停電保持SECS    手動/自動連線
      AND     SM401
      ORB
      OUT     M6002  ; HMI-SECS與上位連線LAMP
32    LD      M1905  ; HMI-PB  SECS-CtlOnline/ Offline
      OR      SM402  ; 初始脈波
      SET     M1906  ; SECS-CtlOnline/ Offline 自保持
35    LDI     M1905  ; HMI-PB  SECS-CtlOnline/ Offline
      LD<=    D9105 K3  ; SECS狀態改變
      MEP
      ORB
      SET     M1907  ; Off-Line自保持
42    LD      M1907  ; Off-Line自保持
      OUT     T1502 K5  ; Off-Line自保持延遲0.5秒
      AND     T1502  ; Off-Line自保持延遲0.5秒
      RST     M1906  ; SECS-CtlOnline/ Offline 自保持
      RST     M1907  ; Off-Line自保持
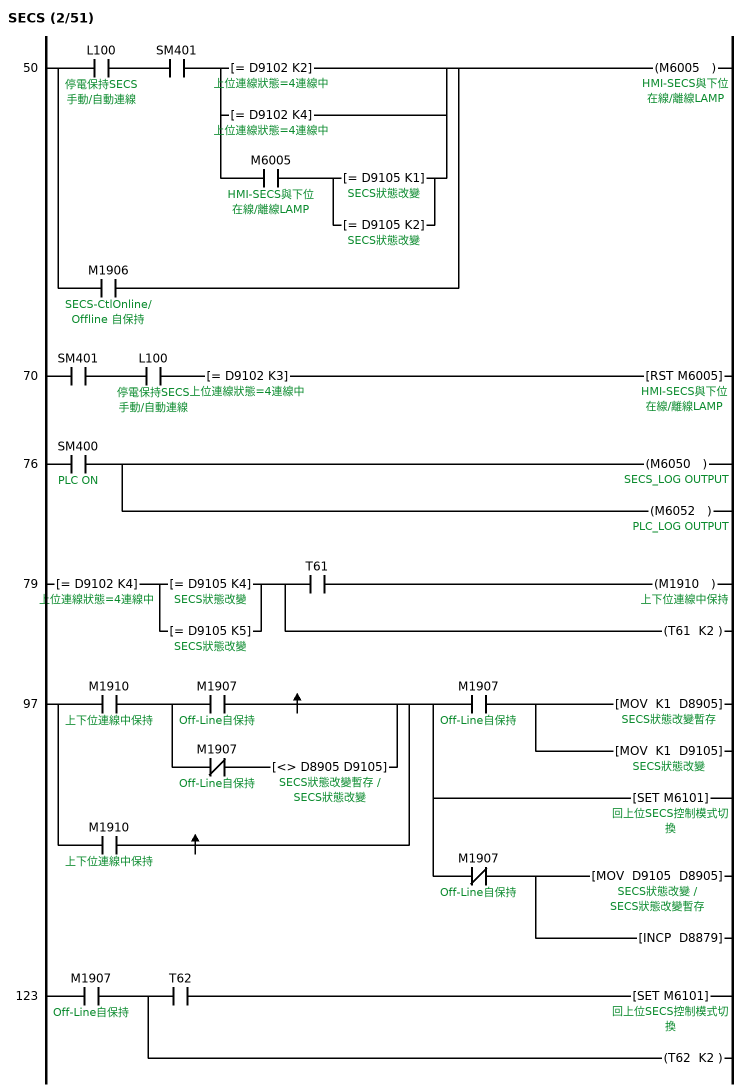
50    LD      L100  ; 停電保持SECS    手動/自動連線
      AND     SM401
      LD=     D9102 K2  ; 上位連線狀態=4連線中
      OR=     D9102 K4  ; 上位連線狀態=4連線中
      LD      M6005  ; HMI-SECS與下位 在線/離線LAMP
      LD=     D9105 K1  ; SECS狀態改變
      OR=     D9105 K2  ; SECS狀態改變
      ANB
      ORB
      ANB
      OR      M1906  ; SECS-CtlOnline/ Offline 自保持
      OUT     M6005  ; HMI-SECS與下位 在線/離線LAMP
70    LD      SM401
      AND     L100  ; 停電保持SECS    手動/自動連線
      AND=    D9102 K3  ; 上位連線狀態=4連線中
      RST     M6005  ; HMI-SECS與下位 在線/離線LAMP
76    LD      SM400  ; PLC ON
      OUT     M6050  ; SECS_LOG OUTPUT
      OUT     M6052  ; PLC_LOG OUTPUT
79    LD=     D9102 K4  ; 上位連線狀態=4連線中
      LD=     D9105 K4  ; SECS狀態改變
      OR=     D9105 K5  ; SECS狀態改變
      ANB
      MPS
      AND     T61
      OUT     M1910  ; 上下位連線中保持
      MPP
      OUT     T61 K2
97    LD      M1910  ; 上下位連線中保持
      LD      M1907  ; Off-Line自保持
      MEP
      LDI     M1907  ; Off-Line自保持
      AND<>   D8905 D9105  ; SECS狀態改變暫存 / SECS狀態改變
      ORB
      ANB
      LD      M1910  ; 上下位連線中保持
      MEP
      ORB
      MPS
      AND     M1907  ; Off-Line自保持
      MOV     K1 D8905
      MOV     K1 D9105
      MPP
      SET     M6101  ; 回上位SECS控制模式切換
      ANI     M1907  ; Off-Line自保持
      MOV     D9105 D8905
      INCP    D8879
123   LD      M1907  ; Off-Line自保持
      MPS
      AND     T62
      SET     M6101  ; 回上位SECS控制模式切換
      MPP
      OUT     T62 K2
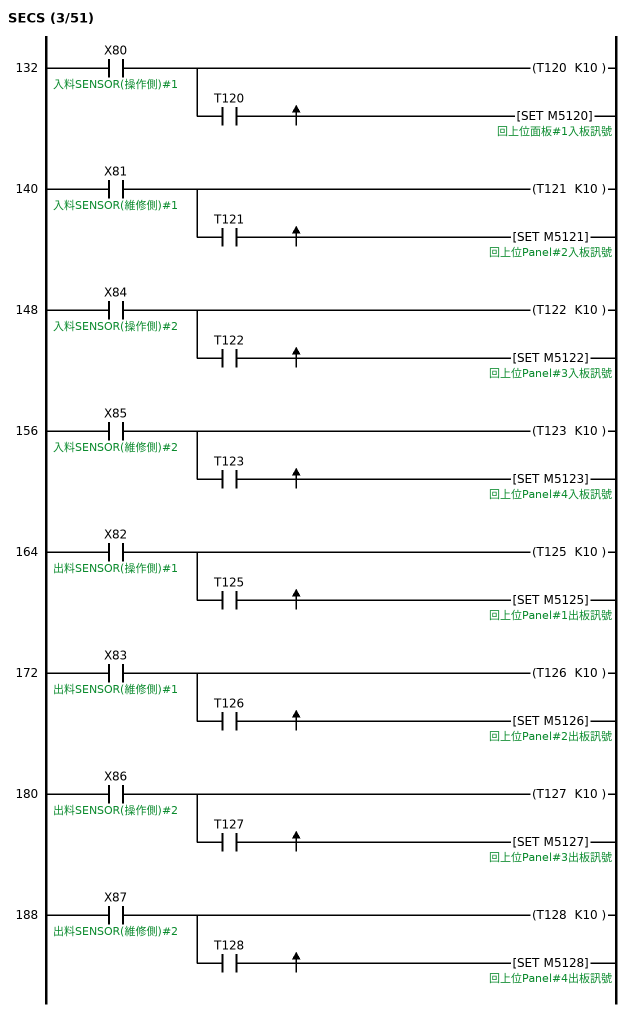
132   LD      X80  ; 入料SENSOR(操作側)#1
      OUT     T120 K10
      AND     T120
      MEP
      SET     M5120  ; 回上位面板#1入板訊號
140   LD      X81  ; 入料SENSOR(維修側)#1
      OUT     T121 K10
      AND     T121
      MEP
      SET     M5121  ; 回上位Panel#2入板訊號
148   LD      X84  ; 入料SENSOR(操作側)#2
      OUT     T122 K10
      AND     T122
      MEP
      SET     M5122  ; 回上位Panel#3入板訊號
156   LD      X85  ; 入料SENSOR(維修側)#2
      OUT     T123 K10
      AND     T123
      MEP
      SET     M5123  ; 回上位Panel#4入板訊號
164   LD      X82  ; 出料SENSOR(操作側)#1
      OUT     T125 K10
      AND     T125
      MEP
      SET     M5125  ; 回上位Panel#1出板訊號
172   LD      X83  ; 出料SENSOR(維修側)#1
      OUT     T126 K10
      AND     T126
      MEP
      SET     M5126  ; 回上位Panel#2出板訊號
180   LD      X86  ; 出料SENSOR(操作側)#2
      OUT     T127 K10
      AND     T127
      MEP
      SET     M5127  ; 回上位Panel#3出板訊號
188   LD      X87  ; 出料SENSOR(維修側)#2
      OUT     T128 K10
      AND     T128
      MEP
      SET     M5128  ; 回上位Panel#4出板訊號
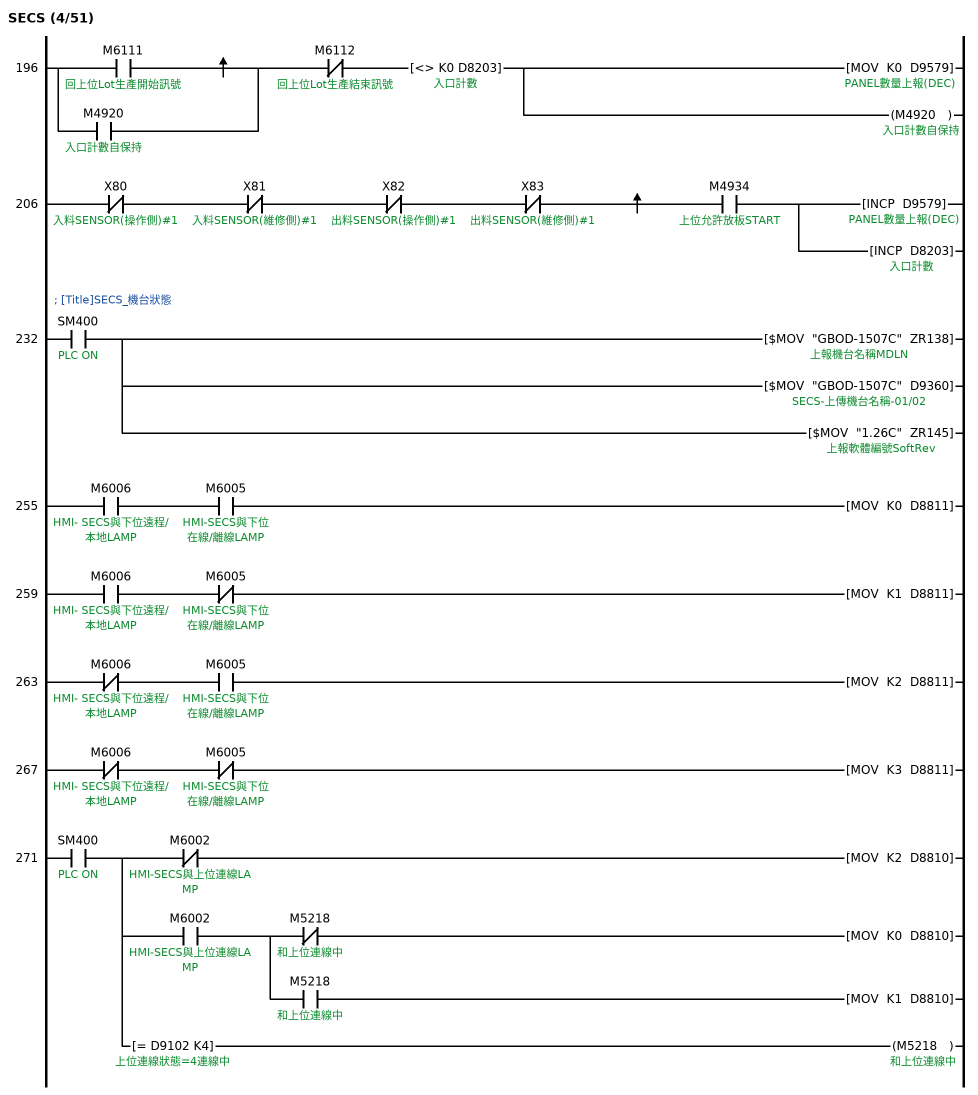
196   LD      M6111  ; 回上位Lot生產開始訊號
      MEP
      OR      M4920  ; 入口計數自保持
      ANI     M6112  ; 回上位Lot生產結束訊號
      AND<>   K0 D8203  ; 入口計數
      MOV     K0 D9579  ; PANEL數量上報(DEC)
      OUT     M4920  ; 入口計數自保持
206   LDI     X80  ; 入料SENSOR(操作側)#1
      ANI     X81  ; 入料SENSOR(維修側)#1
      ANI     X82  ; 出料SENSOR(操作側)#1
      ANI     X83  ; 出料SENSOR(維修側)#1
      MEP
      AND     M4934  ; 上位允許放板START
      INCP    D9579
      INCP    D8203
; [Title]SECS_機台狀態
232   LD      SM400  ; PLC ON
      $MOV    "GBOD-1507C" ZR138  ; 上報機台名稱MDLN
      $MOV    "GBOD-1507C" D9360  ; SECS-上傳機台名稱-01/02
      $MOV    "1.26C" ZR145  ; 上報軟體編號SoftRev
255   LD      M6006  ; HMI- SECS與下位遠程/本地LAMP
      AND     M6005  ; HMI-SECS與下位 在線/離線LAMP
      MOV     K0 D8811
259   LD      M6006  ; HMI- SECS與下位遠程/本地LAMP
      ANI     M6005  ; HMI-SECS與下位 在線/離線LAMP
      MOV     K1 D8811
263   LDI     M6006  ; HMI- SECS與下位遠程/本地LAMP
      AND     M6005  ; HMI-SECS與下位 在線/離線LAMP
      MOV     K2 D8811
267   LDI     M6006  ; HMI- SECS與下位遠程/本地LAMP
      ANI     M6005  ; HMI-SECS與下位 在線/離線LAMP
      MOV     K3 D8811
271   LD      SM400  ; PLC ON
      MPS
      ANI     M6002  ; HMI-SECS與上位連線LAMP
      MOV     K2 D8810
      MRD
      AND     M6002  ; HMI-SECS與上位連線LAMP
      MPS
      ANI     M5218  ; 和上位連線中
      MOV     K0 D8810
      MPP
      AND     M5218  ; 和上位連線中
      MOV     K1 D8810
      MPP
      AND=    D9102 K4  ; 上位連線狀態=4連線中
      OUT     M5218  ; 和上位連線中
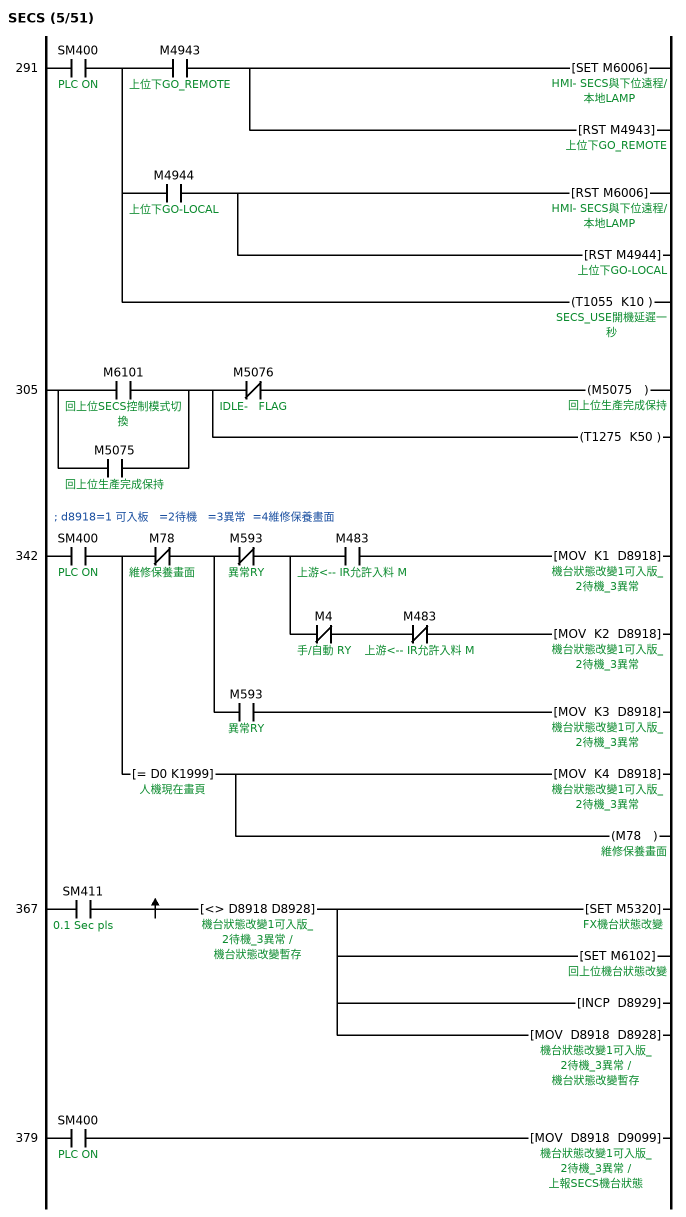
291   LD      SM400  ; PLC ON
      MPS
      AND     M4943  ; 上位下GO_REMOTE
      SET     M6006  ; HMI- SECS與下位遠程/本地LAMP
      RST     M4943  ; 上位下GO_REMOTE
      MRD
      AND     M4944  ; 上位下GO-LOCAL
      RST     M6006  ; HMI- SECS與下位遠程/本地LAMP
      RST     M4944  ; 上位下GO-LOCAL
      MPP
      OUT     T1055 K10  ; SECS_USE開機延遲一秒
305   LD      M6101  ; 回上位SECS控制模式切換
      OR      M5075  ; 回上位生產完成保持
      MPS
      ANI     M5076  ; IDLE-   FLAG
      OUT     M5075  ; 回上位生產完成保持
      MPP
      OUT     T1275 K50
; d8918=1 可入板   =2待機   =3異常  =4維修保養畫面
342   LD      SM400  ; PLC ON
      MPS
      ANI     M78  ; 維修保養畫面
      MPS
      ANI     M593  ; 異常RY
      MPS
      AND     M483  ; 上游<-- IR允許入料 M
      MOV     K1 D8918  ; 機台狀態改變1可入版_2待機_3異常
      MPP
      ANI     M4  ; 手/自動 RY
      ANI     M483  ; 上游<-- IR允許入料 M
      MOV     K2 D8918
      MPP
      AND     M593  ; 異常RY
      MOV     K3 D8918
      MPP
      AND=    D0 K1999  ; 人機現在畫頁
      MOV     K4 D8918
      OUT     M78  ; 維修保養畫面
367   LD      SM411  ; 0.1 Sec pls
      MEP
      AND<>   D8918 D8928  ; 機台狀態改變1可入版_2待機_3異常 / 機台狀態改變暫存
      SET     M5320  ; FX機台狀態改變
      SET     M6102  ; 回上位機台狀態改變
      INCP    D8929
      MOV     D8918 D8928
379   LD      SM400  ; PLC ON
      MOV     D8918 D9099  ; 上報SECS機台狀態
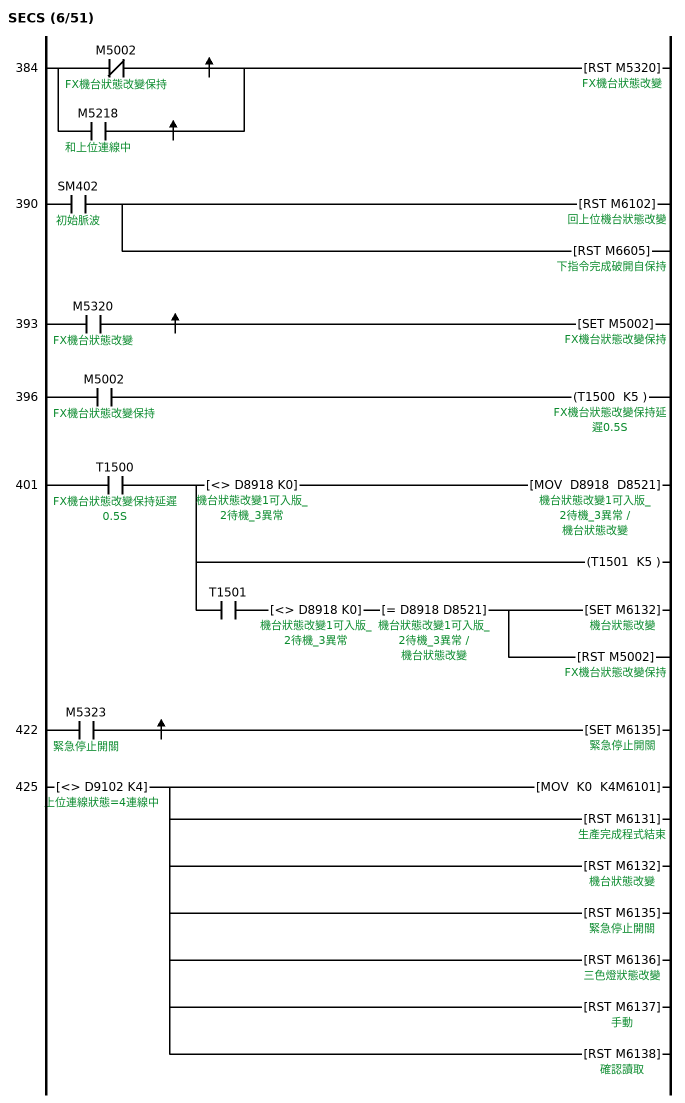
384   LDI     M5002  ; FX機台狀態改變保持
      MEP
      LD      M5218  ; 和上位連線中
      MEP
      ORB
      RST     M5320  ; FX機台狀態改變
390   LD      SM402  ; 初始脈波
      RST     M6102  ; 回上位機台狀態改變
      RST     M6605  ; 下指令完成破開自保持
393   LD      M5320  ; FX機台狀態改變
      MEP
      SET     M5002  ; FX機台狀態改變保持
396   LD      M5002  ; FX機台狀態改變保持
      OUT     T1500 K5  ; FX機台狀態改變保持延遲0.5S
401   LD      T1500  ; FX機台狀態改變保持延遲0.5S
      MPS
      AND<>   D8918 K0  ; 機台狀態改變1可入版_2待機_3異常
      MOV     D8918 D8521  ; 機台狀態改變
      MPP
      OUT     T1501 K5
      AND     T1501
      AND<>   D8918 K0  ; 機台狀態改變1可入版_2待機_3異常
      AND=    D8918 D8521  ; 機台狀態改變1可入版_2待機_3異常 / 機台狀態改變
      SET     M6132  ; 機台狀態改變
      RST     M5002  ; FX機台狀態改變保持
422   LD      M5323  ; 緊急停止開關
      MEP
      SET     M6135  ; 緊急停止開關
425   LD<>    D9102 K4  ; 上位連線狀態=4連線中
      MOV     K0 K4M6101
      RST     M6131  ; 生產完成程式結束
      RST     M6132  ; 機台狀態改變
      RST     M6135  ; 緊急停止開關
      RST     M6136  ; 三色燈狀態改變
      RST     M6137  ; 手動
      RST     M6138  ; 確認讀取
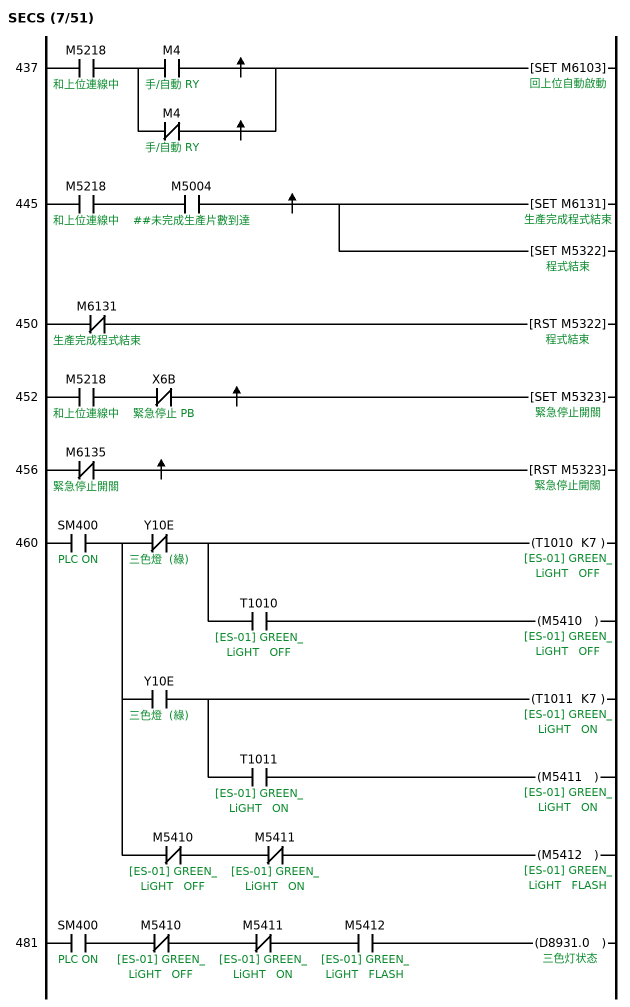
437   LD      M5218  ; 和上位連線中
      LD      M4  ; 手/自動 RY
      MEP
      LDI     M4  ; 手/自動 RY
      MEP
      ORB
      ANB
      SET     M6103  ; 回上位自動啟動
445   LD      M5218  ; 和上位連線中
      AND     M5004  ; ##未完成生產片數到達
      MEP
      SET     M6131  ; 生產完成程式結束
      SET     M5322  ; 程式結束
450   LDI     M6131  ; 生產完成程式結束
      RST     M5322  ; 程式結束
452   LD      M5218  ; 和上位連線中
      ANI     X6B  ; 緊急停止 PB
      MEP
      SET     M5323  ; 緊急停止開關
456   LDI     M6135  ; 緊急停止開關
      MEP
      RST     M5323  ; 緊急停止開關
460   LD      SM400  ; PLC ON
      MPS
      ANI     Y10E  ; 三色燈  (綠)
      OUT     T1010 K7  ; [ES-01] GREEN_  LiGHT   OFF
      AND     T1010  ; [ES-01] GREEN_  LiGHT   OFF
      OUT     M5410  ; [ES-01] GREEN_  LiGHT   OFF
      MRD
      AND     Y10E  ; 三色燈  (綠)
      OUT     T1011 K7  ; [ES-01] GREEN_  LiGHT   ON
      AND     T1011  ; [ES-01] GREEN_  LiGHT   ON
      OUT     M5411  ; [ES-01] GREEN_  LiGHT   ON
      MPP
      ANI     M5410  ; [ES-01] GREEN_  LiGHT   OFF
      ANI     M5411  ; [ES-01] GREEN_  LiGHT   ON
      OUT     M5412  ; [ES-01] GREEN_  LiGHT   FLASH
481   LD      SM400  ; PLC ON
      ANI     M5410  ; [ES-01] GREEN_  LiGHT   OFF
      ANI     M5411  ; [ES-01] GREEN_  LiGHT   ON
      AND     M5412  ; [ES-01] GREEN_  LiGHT   FLASH
      OUT     D8931.0  ; 三色灯状态
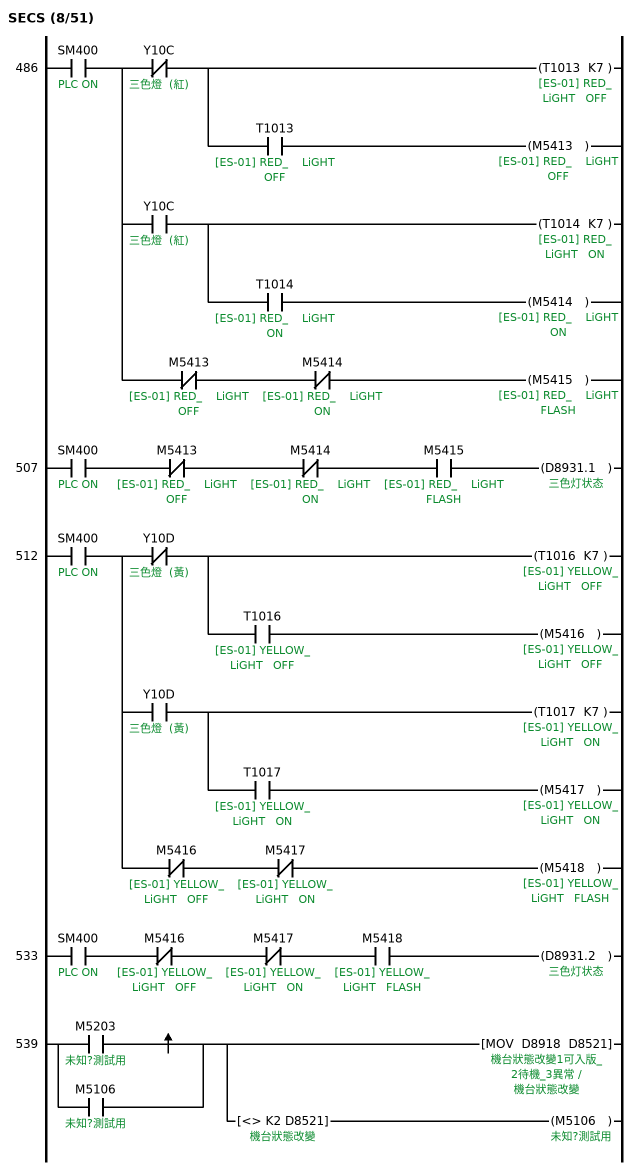
486   LD      SM400  ; PLC ON
      MPS
      ANI     Y10C  ; 三色燈  (紅)
      OUT     T1013 K7  ; [ES-01] RED_    LiGHT   OFF
      AND     T1013  ; [ES-01] RED_    LiGHT   OFF
      OUT     M5413  ; [ES-01] RED_    LiGHT   OFF
      MRD
      AND     Y10C  ; 三色燈  (紅)
      OUT     T1014 K7  ; [ES-01] RED_    LiGHT   ON
      AND     T1014  ; [ES-01] RED_    LiGHT   ON
      OUT     M5414  ; [ES-01] RED_    LiGHT   ON
      MPP
      ANI     M5413  ; [ES-01] RED_    LiGHT   OFF
      ANI     M5414  ; [ES-01] RED_    LiGHT   ON
      OUT     M5415  ; [ES-01] RED_    LiGHT   FLASH
507   LD      SM400  ; PLC ON
      ANI     M5413  ; [ES-01] RED_    LiGHT   OFF
      ANI     M5414  ; [ES-01] RED_    LiGHT   ON
      AND     M5415  ; [ES-01] RED_    LiGHT   FLASH
      OUT     D8931.1  ; 三色灯状态
512   LD      SM400  ; PLC ON
      MPS
      ANI     Y10D  ; 三色燈  (黃)
      OUT     T1016 K7  ; [ES-01] YELLOW_ LiGHT   OFF
      AND     T1016  ; [ES-01] YELLOW_ LiGHT   OFF
      OUT     M5416  ; [ES-01] YELLOW_ LiGHT   OFF
      MRD
      AND     Y10D  ; 三色燈  (黃)
      OUT     T1017 K7  ; [ES-01] YELLOW_ LiGHT   ON
      AND     T1017  ; [ES-01] YELLOW_ LiGHT   ON
      OUT     M5417  ; [ES-01] YELLOW_ LiGHT   ON
      MPP
      ANI     M5416  ; [ES-01] YELLOW_ LiGHT   OFF
      ANI     M5417  ; [ES-01] YELLOW_ LiGHT   ON
      OUT     M5418  ; [ES-01] YELLOW_ LiGHT   FLASH
533   LD      SM400  ; PLC ON
      ANI     M5416  ; [ES-01] YELLOW_ LiGHT   OFF
      ANI     M5417  ; [ES-01] YELLOW_ LiGHT   ON
      AND     M5418  ; [ES-01] YELLOW_ LiGHT   FLASH
      OUT     D8931.2  ; 三色灯状态
539   LD      M5203  ; 未知?測試用
      MEP
      OR      M5106  ; 未知?測試用
      MOV     D8918 D8521
      AND<>   K2 D8521  ; 機台狀態改變
      OUT     M5106  ; 未知?測試用
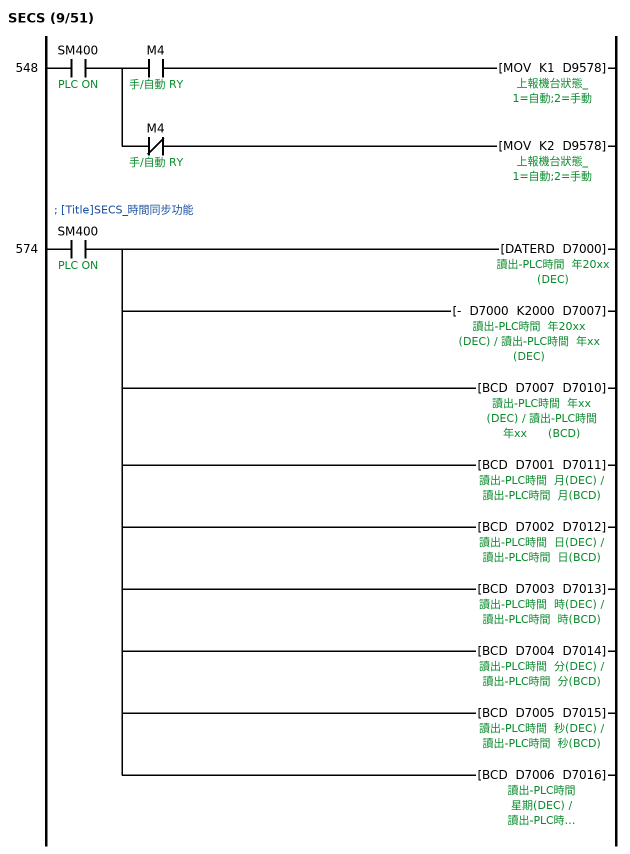
548   LD      SM400  ; PLC ON
      MPS
      AND     M4  ; 手/自動 RY
      MOV     K1 D9578  ; 上報機台狀態_1=自動;2=手動
      MPP
      ANI     M4  ; 手/自動 RY
      MOV     K2 D9578
; [Title]SECS_時間同步功能
574   LD      SM400  ; PLC ON
      DATERD  D7000  ; 讀出-PLC時間  年20xx    (DEC)
      -       D7000 K2000 D7007  ; 讀出-PLC時間  年xx      (DEC)
      BCD     D7007 D7010  ; 讀出-PLC時間  年xx      (BCD)
      BCD     D7001 D7011  ; 讀出-PLC時間  月(DEC) / 讀出-PLC時間  月(BCD)
      BCD     D7002 D7012  ; 讀出-PLC時間  日(DEC) / 讀出-PLC時間  日(BCD)
      BCD     D7003 D7013  ; 讀出-PLC時間  時(DEC) / 讀出-PLC時間  時(BCD)
      BCD     D7004 D7014  ; 讀出-PLC時間  分(DEC) / 讀出-PLC時間  分(BCD)
      BCD     D7005 D7015  ; 讀出-PLC時間  秒(DEC) / 讀出-PLC時間  秒(BCD)
      BCD     D7006 D7016  ; 讀出-PLC時間  星期(DEC) / 讀出-PLC時間  星期(BCD)
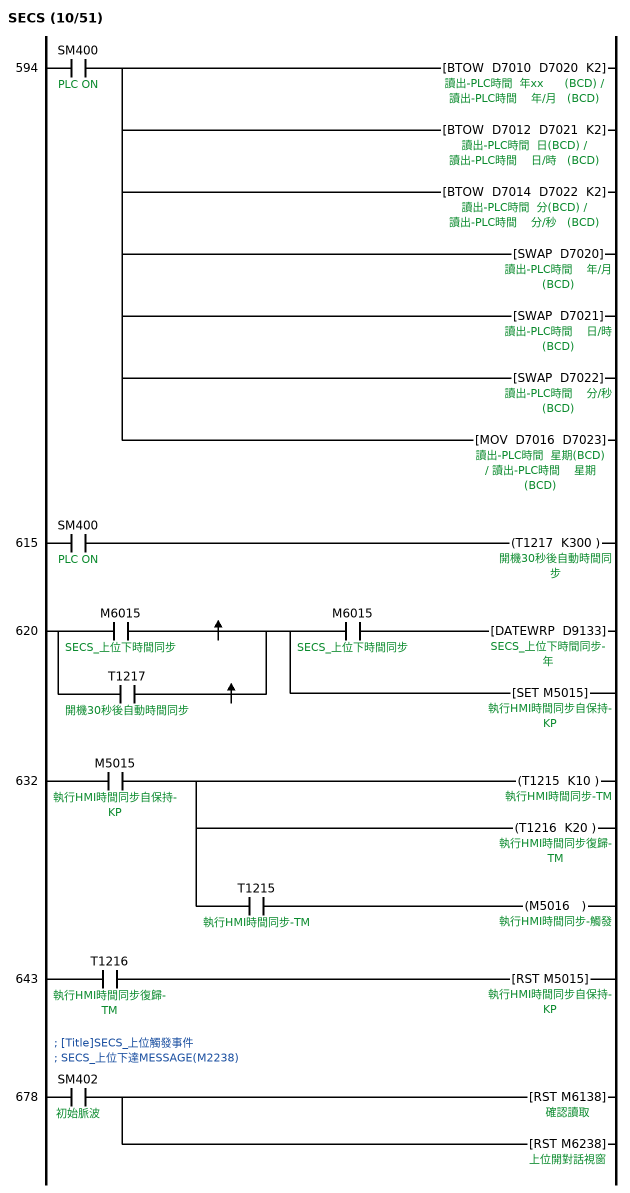
594   LD      SM400  ; PLC ON
      BTOW    D7010 D7020 K2  ; 讀出-PLC時間    年/月   (BCD)
      BTOW    D7012 D7021 K2  ; 讀出-PLC時間    日/時   (BCD)
      BTOW    D7014 D7022 K2  ; 讀出-PLC時間    分/秒   (BCD)
      SWAP    D7020
      SWAP    D7021
      SWAP    D7022
      MOV     D7016 D7023  ; 讀出-PLC時間    星期    (BCD)
615   LD      SM400  ; PLC ON
      OUT     T1217 K300  ; 開機30秒後自動時間同步
620   LD      M6015  ; SECS_上位下時間同步
      MEP
      LD      T1217  ; 開機30秒後自動時間同步
      MEP
      ORB
      MPS
      AND     M6015  ; SECS_上位下時間同步
      DATEWRP D9133  ; SECS_上位下時間同步-年
      MPP
      SET     M5015  ; 執行HMI時間同步自保持-KP
632   LD      M5015  ; 執行HMI時間同步自保持-KP
      OUT     T1215 K10  ; 執行HMI時間同步-TM
      OUT     T1216 K20  ; 執行HMI時間同步復歸-TM
      AND     T1215  ; 執行HMI時間同步-TM
      OUT     M5016  ; 執行HMI時間同步-觸發
643   LD      T1216  ; 執行HMI時間同步復歸-TM
      RST     M5015  ; 執行HMI時間同步自保持-KP
; [Title]SECS_上位觸發事件
; SECS_上位下達MESSAGE(M2238)
678   LD      SM402  ; 初始脈波
      RST     M6138  ; 確認讀取
      RST     M6238  ; 上位開對話視窗
